  GVL_CAM.Control[nAxis].MotionFunction       := ADR(GVL_CAM.MotionFunction);
  GVL_CAM.Control[nAxis].MotionFunctionPoint  := ADR(GVL_CAM.MotionFunctionPoint);
END_FOR
//-----------------------------------------------------------------------------------------------------------------
// assign dataflow/
//-----------------------------------------------------------------------------------------------------------------
//-----------------------------------------------------------------------------------------------------------------
// /INIT
//-----------------------------------------------------------------------------------------------------------------
CASE eInit
OF
  E_PROGRESS.PROGRESS_INVALID:
    FOR nAxis := 1 TO PLC_CONSTANT.MAX_AXIS
    DO
      GVL_MSG_AXIS.MessageLevelAxisCam[nAxis] := E_MessageType.eMessageVerbose;//GVL_MSG.MessageLevel;
    END_FOR
    nAxisInit                                 := 1;
    eInit                                     := E_PROGRESS.PROGRESS_INIT;
  //-----------------------------------------------------------------------------
  //-----------------------------------------------------------------------------
  E_PROGRESS.PROGRESS_INIT:
    stMsg.eType                               := E_MessageType.eMessageInfo;
    stMsg.eDevice                             := e_Device.Device_Main;
    stMsg.eSubdevice                          := e_SubDevice.MainInit;
    stMsg.iErrorNumber                        := MAX_AXIS;
    stMsg.sText                               := concat('CAM.eInit: ', TO_STRING(eInit));
    f_MessageSet(stMsg);

    eInit                                     := E_PROGRESS.PROGRESS_BUSY;
  //-----------------------------------------------------------------------------
  //-----------------------------------------------------------------------------
  E_PROGRESS.PROGRESS_BUSY:
    eInit                                     := E_PROGRESS.PROGRESS_PREPARE;
  //-----------------------------------------------------------------------------
  //-----------------------------------------------------------------------------
  E_PROGRESS.PROGRESS_PREPARE:
    stMsg.eType                               := E_MessageType.eMessageVerbose;
    stMsg.eDevice                             := e_Device.Camming;
    stMsg.eSubdevice                          := e_SubDevice.CamStartUp;
    stMsg.iErrorNumber                        := nAxisInit;
    stMsg.sText                               := concat('AxisInit: ', TO_STRING(nAxisInit));

    IF (GVL_MSG_AXIS.MessageLevelAxisCam[nAxisInit] = E_MessageType.eMessageVerbose)
    THEN
      f_MessageSet(stMsg);
    END_IF

    GVL_CAM.Ctrl[nAxisInit].eCmd              := E_AXIS_CTRL.AXIS_NULL;
    eInit                                     := E_PROGRESS.PROGRESS_STARTUP;


  E_PROGRESS.PROGRESS_STARTUP:
    GVL_CAM.Ctrl[nAxisInit].eCmd              := E_AXIS_CTRL.AXIS_INIT;

    IF (GVL_CAM.State[nAxisInit].eState = E_AXIS_STATE.AXIS_INIT + E_PROGRESS.PROGRESS_ERROR)
    THEN
      eInit                                   := E_PROGRESS.PROGRESS_ERROR;

      stMsg.eType                             := E_MessageType.eMessageError;
      stMsg.eDevice                           := e_Device.Camming;
      stMsg.eSubdevice                        := e_SubDevice.CamStartUp;
      stMsg.iErrorNumber                      := nAxisInit;

      stMsg.sText                             := concat('CAM.eInit ERROR at Index: ', TO_STRING(nAxisInit));
      f_MessageSet(stMsg);

    ELSIF (GVL_CAM.State[nAxisInit].eState = E_AXIS_STATE.AXIS_INIT + E_PROGRESS.PROGRESS_DONE)
    THEN
      eInit                                   := E_PROGRESS.PROGRESS_CHECK;
    END_IF


  E_PROGRESS.PROGRESS_CHECK:
    IF (nAxisInit > PLC_CONSTANT.MAX_AXIS-1)
    THEN
      eInit                                   := E_PROGRESS.PROGRESS_DONE;

      stMsg.eType                             := E_MessageType.eMessageInfo;
      stMsg.eDevice                           := e_Device.Device_Cam;
      stMsg.eSubdevice                        := e_SubDevice.CamStartUp;
      stMsg.iErrorNumber                      := MAX_AXIS;

      stMsg.sText                             := concat('CAM.eInit: ', TO_STRING(eInit));
      f_MessageSet(stMsg);

      FOR nAxis := 1 TO PLC_CONSTANT.MAX_AXIS
      DO
        GVL_MSG_AXIS.MessageLevelAxisCam[nAxis]  := GVL_MSG_AXIS.MessageLevel;
      END_FOR
    ELSE
      nAxisInit                               := nAxisInit + 1;
      eInit                                   := E_PROGRESS.PROGRESS_PREPARE;
    END_IF
END_CASE
//-----------------------------------------------------------------------------------------------------------------
// INIT
//-----------------------------------------------------------------------------------------------------------------
//-----------------------------------------------------------------------------------------------------------------
// /cyclic
//-----------------------------------------------------------------------------------------------------------------
IF (eInit <> E_PROGRESS.PROGRESS_ERROR)
THEN
  FOR nAxis := 1 TO PLC_CONSTANT.MAX_AXIS
  DO
      GVL_CAM.Control[nAxis].Cycle();
  END_FOR
END_IF
//-----------------------------------------------------------------------------------------------------------------
// cyclic/
//-----------------------------------------------------------------------------------------------------------------

END_PROGRAM

// ---- PLC_MOTION/NCI/class/FB_NciChannelCtrl.TcPOU
(*
-------------------------------------------------------------------------------
	NCI Channel Control

  2020/05/20  HAUD  0.1     kinematic and NCI separation
  2022/10/22  HAUD  0.2     PLC_OPEN_DRIVE adaption
  2023/12/29  HAUD  0.3     PLC_STATE_DRIVE adaption
-------------------------------------------------------------------------------
*)

// This SOFTWARE is provided as an Exemple by THE PROVIDER "as is" and "with all faults." THE PROVIDER makes no 
// representations or warranties of any kind concerning the safety, suitability, lack of viruses, inaccuracies, 
// typographical errors, or other harmful components of this SOFTWARE. There are inherent dangers in the use of 
// any software, and you are solely responsible for determining whether this SOFTWARE is compatible with your 
// equipment and other software installed on your equipment. You are also solely responsible for the protection 
// of your equipment and backup of your data, and THE PROVIDER will not be liable for any damages you may suffer 
// in connection with using, modifying, or distributing this SOFTWARE.

FUNCTION_BLOCK FB_NciChannelCtrl EXTENDS FB_NciChannel IMPLEMENTS I_Nci_Ctrl
VAR
  _stChannelRef         : ST_NciChannel_Ref;
  _nChnId               : UINT;

  _eCtrl,
  _eCtrlOld             : E_NCI_CTRL;

  _eState               : E_NCI_STATE;

  _eInit,
  _eResult,
  _eResultOld           : E_PROGRESS;

  // control and state struct from outside world
  _Ctrl                 : POINTER TO ST_NCI_CTRL;
  _State                : POINTER TO ST_NCI_STATE;

  // M function to fetch for scope/debugging
  _MFuncScope           : POINTER TO ST_NCI_M_FUNC;

  _fPathVelo            : LREAL;
  _nBlockNo             : UDINT;
  _sProgLine            : STRING(100); 
  _nMFunc               : INT;
  _nStateItp            : UINT;
END_VAR

METHOD Check : BOOL
VAR_INST
 
END_VAR

IF NOT SUPER^.Check() THEN RETURN; END_IF

IF NOT (_Ctrl <> 0)
THEN
  _eCheck                     := E_CHECK_STATE.NCI_CTRL_POINTER_INVALID;
  RETURN;
END_IF

IF NOT (_State <> 0)
THEN
  _eCheck                     := E_CHECK_STATE.NCI_STATE_POINTER_INVALID;
  RETURN;
END_IF

IF NOT (_MFuncScope <> 0)
THEN
  _eCheck                     := E_CHECK_STATE.NCI_M_FUNC_POINTER_INVALID;
  RETURN;
END_IF

_eCheck                       := E_CHECK_STATE.CHECK_DONE;
Check                         := TRUE;
END_METHOD

PROPERTY ChnCtrl : pointer to ST_NCI_CTRL
SET
_Ctrl := ChnCtrl;
END_SET
END_PROPERTY

PROPERTY ChnId : udint
GET
ChnId := _NciChannelRef^.NcToPlc.ChnId;
END_GET
END_PROPERTY

PROPERTY ChnState : pointer to ST_NCI_STATE
SET
_State := ChnState;
END_SET
END_PROPERTY

//
//  Cmd
//    - gets state for ctrl
//    - prepare your commands here
//    - init what you have to here
//
//-------------------------------------------------------------------------------------
METHOD PRIVATE Cmd  : E_NCI_STATE
VAR_INPUT
  eCmd      : E_NCI_CTRL;
END_VAR
VAR_INST
  _estate   : E_NCI_STATE;
  _stMsg    : ST_Message;
END_VAR

CASE eCmd
OF
  E_NCI_CTRL.INIT:
    // check axis configuration, clear group, reset Itp
    _eInit := _eResult      := Ctrl_Init(FALSE);
    _eState                 := E_NCI_STATE.INIT;
ELSE
  IF NOT (_eInit = E_PROGRESS.PROGRESS_DONE)
  THEN
    _eResult                := E_PROGRESS.PROGRESS_ERROR;
  
    _stMsg.eType            := E_MessageType.eMessageError;
    _stMsg.eDevice          := E_Device.NciChannelCtrl + (ChnId);
    _stMsg.eSubdevice       := e_Subdevice.NciControl;
    _stMsg.iErrorNumber     := 1;
  
    _stMsg.sText          := 'eInit:';
    _stMsg.sText          := concat(_stMsg.sText, TO_STRING(_eInit));
    _stMsg.sText          := concat(_stMsg.sText, ': ');
    _stMsg.sText          := concat(_stMsg.sText, TO_STRING(_eResult));

    f_MessageSet(_stMsg);

  ELSE
    CASE eCmd
    OF
      E_NCI_CTRL.IDLE:
        _eResult                := Ctrl_Idle(FALSE);
        _eState                 := E_NCI_STATE.IDLE;
    
      E_NCI_CTRL.FEED_TABLE:
        // nothing implemented yet
        _eResult                := E_PROGRESS.PROGRESS_NOT_EXIST;
        _eState                 := E_NCI_STATE.FEED_TABLE;
    
      E_NCI_CTRL.RESET:
        _eResult                := Ctrl_Reset(FALSE);
        _eState                 := E_NCI_STATE.RESET;
    
      E_NCI_CTRL.LOAD_PROG:
        _eResult                := Ctrl_LoadProg(FALSE);
        _eState                 := E_NCI_STATE.LOAD_PROG;
    
      E_NCI_CTRL.BUILD_GROUP:
        _eResult                := Ctrl_BuildGroup(FALSE);
        _eState                 := E_NCI_STATE.BUILD_GROUP;
    
      E_NCI_CTRL.CLEAR_GROUP:
        _eResult                := Ctrl_ClearGroup(FALSE);
        _eState                 := E_NCI_STATE.CLEAR_GROUP;
    
      E_NCI_CTRL.START:
        _eResult                := Ctrl_Start(FALSE);
        _eState                 := E_NCI_STATE.START;
    
      E_NCI_CTRL.STOP:
        _eResult                := Ctrl_Stop(FALSE);
        _eState                 := E_NCI_STATE.STOP;
    
      E_NCI_CTRL.STO_STOP:
        _eResult                := Ctrl_Stop_STO(FALSE);
        _eState                 := E_NCI_STATE.STO_STOP;
    
      E_NCI_CTRL.RESTART_STEP_ON:
        _eResult                := Ctrl_Restart(FALSE);
        _eState                 := E_NCI_STATE.RESTART_STEP_ON;
    
      E_NCI_CTRL.M_FUNC_QUIT:
        _eResult                := Ctrl_ConfirmHsk(FALSE);
        _eState                 := E_NCI_STATE.M_FUNC_QUIT;
    
      E_NCI_CTRL.READ_R_PARA:
        _eResult                := Ctrl_R_Parameter_Rd(FALSE);
        _eState                 := E_NCI_STATE.READ_R_PARA;
    
      E_NCI_CTRL.WRITE_R_PARA:
        _eResult                := Ctrl_R_Parameter_Wrt(FALSE);
        _eState                 := E_NCI_STATE.WRITE_R_PARA;
    ELSE
      _eState                 := E_NCI_STATE.NULL;
  
      IF (eCmd = E_NCI_CTRL.NULL)
      THEN
        _eResult              := E_PROGRESS.PROGRESS_DONE;
      ELSE
        _eResult              := E_PROGRESS.PROGRESS_INVALID;
  
        _stMsg.eType          := E_MessageType.eMessageError;
        _stMsg.eDevice        := E_Device.NciChannelCtrl + (ChnId);
        _stMsg.eSubdevice     := e_Subdevice.NciControl;
        _stMsg.iErrorNumber   := 0;
  
        _stMsg.sText          := 'E_NCI_CTRL.';
        _stMsg.sText          := concat(_stMsg.sText, TO_STRING(eCmd));
        _stMsg.sText          := concat(_stMsg.sText, ': ');
        _stMsg.sText          := concat(_stMsg.sText, TO_STRING(_eResult));
  
        f_MessageSet(_stMsg);
      END_IF
    END_CASE
  END_IF
END_CASE


Cmd                         := _eState;
END_METHOD

METHOD PRIVATE Ctrl_BuildGroup : E_PROGRESS
VAR_INPUT
  Execute           : BOOL;
END_VAR
VAR_INST
  _eJobResult,
  _eState           : E_PROGRESS;
END_VAR
IF NOT Check() THEN Ctrl_BuildGroup := E_PROGRESS.PROGRESS_ERROR; RETURN; END_IF
IF NOT Execute THEN _eState := E_PROGRESS.PROGRESS_INIT; END_IF

CASE _eState
OF
  E_PROGRESS.PROGRESS_INIT:
    IF Execute 
    THEN
      _eJobResult                   := BuilDGroup(FALSE);
      _eState                       := E_PROGRESS.PROGRESS_BUSY;
    END_IF
END_CASE
CASE _eState
OF
  E_PROGRESS.PROGRESS_BUSY:
    _eJobResult                     := BuilDGroup(TRUE);

    IF (_eJobResult = E_PROGRESS.PROGRESS_ERROR)
    THEN
      BuilDGroup(FALSE);
      _eState                       := E_PROGRESS.PROGRESS_ERROR;

    ELSIF (_eJobResult = E_PROGRESS.PROGRESS_DONE)
    THEN
      BuilDGroup(FALSE);
      _eState                       := E_PROGRESS.PROGRESS_STARTUP;
    END_IF
END_CASE
CASE _eState
OF
  E_PROGRESS.PROGRESS_STARTUP:
    _eState                         := E_PROGRESS.PROGRESS_PREPARE;
END_CASE
CASE _eState
OF
  E_PROGRESS.PROGRESS_PREPARE:
    _eState                         := E_PROGRESS.PROGRESS_CHECK;
END_CASE
CASE _eState
OF
  E_PROGRESS.PROGRESS_CHECK:
    _eState                         := E_PROGRESS.PROGRESS_OCCUPIED;
END_CASE
CASE _eState
OF
  E_PROGRESS.PROGRESS_OCCUPIED:
    _eState                         := E_PROGRESS.PROGRESS_WORKING;
END_CASE
CASE _eState
OF
  E_PROGRESS.PROGRESS_WORKING:
    _eState                         := E_PROGRESS.PROGRESS_DONE;
END_CASE

Ctrl_BuildGroup                      := _eState;
END_METHOD

METHOD PRIVATE Ctrl_ClearGroup : E_PROGRESS
VAR_INPUT
  Execute           : BOOL;
END_VAR
VAR_INST
  _eJobResult,
  _eState           : E_PROGRESS;
END_VAR
IF NOT Check() THEN Ctrl_ClearGroup := E_PROGRESS.PROGRESS_ERROR; RETURN; END_IF
IF NOT Execute THEN _eState := E_PROGRESS.PROGRESS_INIT; END_IF

CASE _eState
OF
  E_PROGRESS.PROGRESS_INIT:
    IF Execute 
    THEN
      _eJobResult                           := ClearGroup(FALSE);
      _eState                               := E_PROGRESS.PROGRESS_BUSY;
    END_IF

  E_PROGRESS.PROGRESS_BUSY:
    _eJobResult                             := ClearGroup(TRUE);
    IF (_eJobResult = E_PROGRESS.PROGRESS_ERROR)
    THEN
      ClearGroup(FALSE);
      _eState                               := E_PROGRESS.PROGRESS_ERROR;

    ELSIF (_eJobResult = E_PROGRESS.PROGRESS_DONE)
    THEN
      ClearGroup(FALSE);
      _eJobResult                           := ItpReset(FALSE);
      _eState                               := E_PROGRESS.PROGRESS_STARTUP;
    END_IF

  E_PROGRESS.PROGRESS_STARTUP:
    _eJobResult                             := ItpReset(TRUE);
    IF (_eJobResult = E_PROGRESS.PROGRESS_ERROR)
    THEN
      ItpReset(FALSE);
      _eState                               := E_PROGRESS.PROGRESS_ERROR;

    ELSIF (_eJobResult = E_PROGRESS.PROGRESS_DONE)
    THEN
      ItpReset(FALSE);
      _eState                               := E_PROGRESS.PROGRESS_PREPARE;
    END_IF

  E_PROGRESS.PROGRESS_PREPARE:
    IF (_NciChannelRef^.NcToPlc.HskMFuncReq = 0)
    THEN
      _eState                               := E_PROGRESS.PROGRESS_DONE;
    ELSE
      _NciChannelRef^.PlcToNc.MFuncGranted  := 0;
      _eState                               := E_PROGRESS.PROGRESS_CHECK;
    END_IF

  E_PROGRESS.PROGRESS_CHECK:
      _NciChannelRef^.PlcToNc.MFuncGranted  := 1;
      _eState                               := E_PROGRESS.PROGRESS_PREPARE;

  E_PROGRESS.PROGRESS_DONE:
    _NciChannelRef^.PlcToNc.MFuncGranted    := 0;
END_CASE


Ctrl_ClearGroup                             := _eState;
END_METHOD

METHOD PRIVATE Ctrl_ConfirmHsk : E_PROGRESS
VAR_INPUT
  Execute           : BOOL;
END_VAR
VAR_INST
  _eJobResult,
  _eState           : E_PROGRESS;
END_VAR
IF NOT Check() THEN Ctrl_ConfirmHsk := E_PROGRESS.PROGRESS_ERROR; RETURN; END_IF
IF NOT Execute THEN _eState := E_PROGRESS.PROGRESS_INIT; END_IF

CASE _eState
OF
  E_PROGRESS.PROGRESS_INIT:
    IF Execute 
    THEN
      _eJobResult                         := ConfirmHSK(FALSE);
      _eState                             := E_PROGRESS.PROGRESS_BUSY;
    END_IF
END_CASE
CASE _eState
OF

  E_PROGRESS.PROGRESS_BUSY:
    _eJobResult                           := ConfirmHSK(TRUE);

    IF (_eJobResult = E_PROGRESS.PROGRESS_ERROR)
    THEN
      ConfirmHSK(FALSE);
      _eState                             := E_PROGRESS.PROGRESS_ERROR;

    ELSIF (_eJobResult = E_PROGRESS.PROGRESS_DONE)
    THEN
      ConfirmHSK(FALSE);
      _eState                             := E_PROGRESS.PROGRESS_PREPARE;
    END_IF
END_CASE
CASE _eState
OF
  E_PROGRESS.PROGRESS_PREPARE:
    _eState                               := E_PROGRESS.PROGRESS_DONE;
    // update connected struct data
    _MFuncScope^.FastMFuncMask            := _NciChannelRef^.NcToPlc.FastMFuncMask;
    _MFuncScope^.HskMFuncNo               := _NciChannelRef^.NcToPlc.HskMFuncNo;
    _MFuncScope^.HskMFuncReq              := _NciChannelRef^.NcToPlc.HskMFuncReq;
    _MFuncScope^.HFuncValue               := _NciChannelRef^.NcToPlc.HFuncValue;
    _MFuncScope^.MFuncGranted             := _NciChannelRef^.PlcToNc.MFuncGranted;
END_CASE

Ctrl_ConfirmHsk                            := _eState;
END_METHOD

METHOD PRIVATE Ctrl_Idle : E_PROGRESS
VAR_INPUT
  Execute           : BOOL;
END_VAR
VAR_INST
  _eJobResult,
  _eState           : E_PROGRESS;

  _nErr             : DWORD;
  _NciAxisIds       : ARRAY[1..8] OF DWORD;

  _stMsg            : ST_Message;
END_VAR
IF NOT Check() THEN Ctrl_Idle := E_PROGRESS.PROGRESS_ERROR; RETURN; END_IF
IF NOT Execute THEN _eState := E_PROGRESS.PROGRESS_INIT; END_IF

CASE _eState
OF
  E_PROGRESS.PROGRESS_INIT:
    IF Execute 
    THEN
      _eJobResult                         := ItpReset(FALSE);
      _eState                             := E_PROGRESS.PROGRESS_BUSY;
    END_IF
END_CASE
CASE _eState
OF
  E_PROGRESS.PROGRESS_BUSY:
    IF (_NciChannelRef^.NcToPlc.ItpState <> Tc2_NCI.NCI_INTERPRETER_IDLE)
    THEN
      _eState                             := E_PROGRESS.PROGRESS_STARTUP;
    ELSE
      IF (_NciChannelRef^.PlcToNc.ChnAxesOvr > 0) AND NOT
         (_NciChannelRef^.NcToPlc.ChnState.8)
      THEN
        _eState                           := E_PROGRESS.PROGRESS_PREPARE;
      END_IF
    END_IF
END_CASE
CASE _eState
OF
  E_PROGRESS.PROGRESS_STARTUP:
    _eJobResult                           := ItpReset(TRUE);
    IF (_eJobResult = E_PROGRESS.PROGRESS_ERROR)
    THEN
      ItpReset(FALSE);
      _eState                             := E_PROGRESS.PROGRESS_ERROR;

    ELSIF (_eJobResult = E_PROGRESS.PROGRESS_DONE)
    THEN
      ItpReset(FALSE);
      _eState                             := E_PROGRESS.PROGRESS_PREPARE;
    END_IF

  E_PROGRESS.PROGRESS_PREPARE:
    _NciChannelRef^.PlcToNc.MFuncGranted  := 0;
    _eState                               := E_PROGRESS.PROGRESS_CHECK;

END_CASE
CASE _eState
OF
  E_PROGRESS.PROGRESS_CHECK:
    _nErr                                 := ItpGetGroupAxisIds(_NciAxisIds, _NciChannelRef^.NcToPlc);

    IF (_NciChannelRef^.NcToPlc.HskMFuncReq = 0)
    THEN
      IF (_nErr <> 0)
      THEN
        _eState                           := E_PROGRESS.PROGRESS_ERROR;
        _stMsg.eType                      := E_MessageType.eMessageError;
        _stMsg.eDevice                    := ChannelDevice;
        _stMsg.eSubdevice                 := e_Subdevice.NciIdle;
        _stMsg.iErrorNumber               := _nErr;
        _stMsg.sText                      := concat('ItpGetGroupAxisIds Error: ', TO_STRING(_nErr));

        f_MessageSet(_stMsg);
      ELSE
        _eState                           := E_PROGRESS.PROGRESS_DONE;
      END_IF
    ELSE
      _eState                             := E_PROGRESS.PROGRESS_STARTUP;
    END_IF
END_CASE

Ctrl_Idle                                := _eState;
END_METHOD

METHOD Ctrl_Init : E_PROGRESS
VAR_INPUT
  Execute           : BOOL;
END_VAR
VAR_INST
  _eJobResult,
  _eState           : E_PROGRESS;
  _rValue           : LREAL;
  _udiErr           : UDINT;

  _nErr             : DWORD;
  _NciAxisIds       : ARRAY[1..8] OF DWORD;

  _stMsg            : ST_Message;
END_VAR
IF NOT Check() THEN _eState := E_PROGRESS.PROGRESS_ERROR; END_IF
IF NOT Execute THEN _eState := E_PROGRESS.PROGRESS_INIT; END_IF

CASE _eState
OF
  E_PROGRESS.PROGRESS_INIT:
    IF Execute 
    THEN
      memset(ADR(_stMsg),0,SIZEOF(_stMsg));
      _udiErr                       := 0;
      _rValue                       := 0;
      _eState                       := E_PROGRESS.PROGRESS_BUSY;
    END_IF
END_CASE
CASE _eState
OF
  E_PROGRESS.PROGRESS_BUSY:
    IF NOT (_stCfgAxes^.nXAxisId > 0) OR
       NOT (_stCfgAxes^.nYAxisId > 0) OR
       NOT (_stCfgAxes^.nZAxisId > 0)
    THEN
      _eState                       := E_PROGRESS.PROGRESS_OCCUPIED;

      _stMsg.eType                  := E_MessageType.eMessageWarning;
      _stMsg.eDevice                := ChannelDevice;
      _stMsg.eSubdevice             := e_Subdevice.NciStartUp;
      _stMsg.iErrorNumber           := _eState;
      _stMsg.sText                  := concat('Init NCI channel AxisConfig: ', TO_STRING(_eState));

      f_MessageSet(_stMsg);
    ELSE
      _eJobResult                   := ItpReset(FALSE);
      _eState                       := E_PROGRESS.PROGRESS_STARTUP;
    END_IF
END_CASE
CASE _eState
OF
  E_PROGRESS.PROGRESS_STARTUP:
    _eJobResult                     := ItpReset(TRUE);
    IF (_eJobResult = E_PROGRESS.PROGRESS_ERROR)
    THEN
      _eState                       := E_PROGRESS.PROGRESS_ERROR;
    ELSIF (_eJobResult = E_PROGRESS.PROGRESS_DONE)
    THEN
      _eJobResult                   := ItpReset  (FALSE);
      _eJobResult                   := ClearGroup(FALSE);
      _eState                       := E_PROGRESS.PROGRESS_PREPARE;
    END_IF
END_CASE
CASE _eState
OF
  E_PROGRESS.PROGRESS_PREPARE:
    _eJobResult                     := ClearGroup(TRUE);
    IF (_eJobResult = E_PROGRESS.PROGRESS_ERROR)
    THEN
      _eState                       := E_PROGRESS.PROGRESS_ERROR;
    ELSIF (_eJobResult = E_PROGRESS.PROGRESS_DONE)
    THEN
      _eJobResult                   := ClearGroup(FALSE);
      _eState                       := E_PROGRESS.PROGRESS_CHECK;
    END_IF

END_CASE
CASE _eState
OF
  E_PROGRESS.PROGRESS_CHECK:
    _eState                         := E_PROGRESS.PROGRESS_WORKING;
END_CASE
CASE _eState
OF
  E_PROGRESS.PROGRESS_OCCUPIED:
    IF (_stCfgAxes^.nXAxisId > 0) AND
       (_stCfgAxes^.nYAxisId > 0) AND
       (_stCfgAxes^.nZAxisId > 0)
    THEN
      _eState                       := E_PROGRESS.PROGRESS_STARTUP;

      _stMsg.eType                  := E_MessageType.eMessageInfo;
      _stMsg.eDevice                := ChannelDevice;
      _stMsg.eSubdevice             := e_Subdevice.NciStartUp;
      _stMsg.iErrorNumber           := _eState;
      _stMsg.sText                  := concat('Init NCI channel AxisConfig: ', TO_STRING(_eState));

      IF (_MessageLevel < E_MessageType.eMessageError)
      THEN
        f_MessageSet(_stMsg);
      END_IF
    END_IF
END_CASE
CASE _eState
OF
  E_PROGRESS.PROGRESS_WORKING:
    _eState                         := E_PROGRESS.PROGRESS_DONE;
END_CASE

Ctrl_Init                           := _eState;
END_METHOD

METHOD PRIVATE Ctrl_LoadProg : E_PROGRESS
VAR_INPUT
  Execute           : BOOL;
END_VAR
VAR_INST
  _eJobResult,
  _eState           : E_PROGRESS;
END_VAR
IF NOT Check() THEN Ctrl_LoadProg := E_PROGRESS.PROGRESS_ERROR; RETURN; END_IF
IF NOT Execute THEN _eState := E_PROGRESS.PROGRESS_INIT; END_IF

CASE _eState
OF
  E_PROGRESS.PROGRESS_INIT:
    IF Execute 
    THEN
      _eJobResult                         := LoadProg(FALSE);
      _eState                             := E_PROGRESS.PROGRESS_BUSY;
    END_IF

  E_PROGRESS.PROGRESS_BUSY:
    _NciChannelRef^.PlcToNc.MFuncGranted  := 0;
    _eJobResult                           := LoadProg(TRUE);

    IF (_eJobResult = E_PROGRESS.PROGRESS_ERROR)
    THEN
      LoadProg(FALSE);
      _eState                             := E_PROGRESS.PROGRESS_ERROR;

    ELSIF (_eJobResult = E_PROGRESS.PROGRESS_DONE)
    THEN
      LoadProg(FALSE);
      _eState                             := E_PROGRESS.PROGRESS_DONE;
    END_IF
END_CASE

Ctrl_LoadProg                      := _eState;
END_METHOD

METHOD PRIVATE Ctrl_R_Parameter_Rd : E_PROGRESS
VAR_INPUT
  Execute           : BOOL;
END_VAR
VAR_INST
  _eJobResult,
  _eState           : E_PROGRESS;
END_VAR
IF NOT Check() THEN Ctrl_R_Parameter_Rd := E_PROGRESS.PROGRESS_ERROR; RETURN; END_IF
IF NOT Execute THEN _eState := E_PROGRESS.PROGRESS_INIT; END_IF

CASE _eState
OF
  E_PROGRESS.PROGRESS_INIT:
    IF Execute 
    THEN
      _eJobResult                         := ReadRParams(FALSE);
      _eState                             := E_PROGRESS.PROGRESS_BUSY;
    END_IF

  E_PROGRESS.PROGRESS_BUSY:
    _NciChannelRef^.PlcToNc.MFuncGranted  := 0;
    _eJobResult                           := ReadRParams(TRUE);

    IF (_eJobResult = E_PROGRESS.PROGRESS_ERROR)
    THEN
      ReadRParams(FALSE);
      _eState                             := E_PROGRESS.PROGRESS_ERROR;

    ELSIF (_eJobResult = E_PROGRESS.PROGRESS_DONE)
    THEN
      ReadRParams(FALSE);
      _eState                             := E_PROGRESS.PROGRESS_STARTUP;
    END_IF
END_CASE
CASE _eState
OF
  E_PROGRESS.PROGRESS_STARTUP:
    _NciChannelRef^.PlcToNc.MFuncGranted  := 1;
    _eState                               := E_PROGRESS.PROGRESS_PREPARE;

  E_PROGRESS.PROGRESS_PREPARE:
    _NciChannelRef^.PlcToNc.MFuncGranted  := 0;
    _eState                               := E_PROGRESS.PROGRESS_DONE;
END_CASE

Ctrl_R_Parameter_Rd                       := _eState;
END_METHOD

METHOD PRIVATE Ctrl_R_Parameter_Wrt : E_PROGRESS
VAR_INPUT
  Execute           : BOOL;
END_VAR
VAR_INST
  _eJobResult,
  _eState           : E_PROGRESS;
END_VAR
IF NOT Check() THEN Ctrl_R_Parameter_Wrt := E_PROGRESS.PROGRESS_ERROR; RETURN; END_IF
IF NOT Execute THEN _eState := E_PROGRESS.PROGRESS_INIT; END_IF

CASE _eState
OF
  E_PROGRESS.PROGRESS_INIT:
    IF Execute 
    THEN
      _eJobResult                         := WriteRParams(FALSE);
      _eState                             := E_PROGRESS.PROGRESS_BUSY;
    END_IF

  E_PROGRESS.PROGRESS_BUSY:
    _NciChannelRef^.PlcToNc.MFuncGranted  := 0;
    _eJobResult                           := WriteRParams(TRUE);

    IF (_eJobResult = E_PROGRESS.PROGRESS_ERROR)
    THEN
      WriteRParams(FALSE);
      _eState                             := E_PROGRESS.PROGRESS_ERROR;

    ELSIF (_eJobResult = E_PROGRESS.PROGRESS_DONE)
    THEN
      WriteRParams(FALSE);
      _eState                             := E_PROGRESS.PROGRESS_STARTUP;
    END_IF
END_CASE
CASE _eState
OF
  E_PROGRESS.PROGRESS_STARTUP:
    _NciChannelRef^.PlcToNc.MFuncGranted  := 1;
    _eState                               := E_PROGRESS.PROGRESS_PREPARE;

  E_PROGRESS.PROGRESS_PREPARE:
    _NciChannelRef^.PlcToNc.MFuncGranted  := 0;
    _eState                               := E_PROGRESS.PROGRESS_DONE;
END_CASE

Ctrl_R_Parameter_Wrt                      := _eState;
END_METHOD

METHOD PRIVATE Ctrl_Reset : E_PROGRESS
VAR_INPUT
  Execute           : BOOL;
END_VAR
VAR_INST
  _eJobResult,
  _eState           : E_PROGRESS;
END_VAR
IF NOT Check() THEN Ctrl_Reset := E_PROGRESS.PROGRESS_ERROR; RETURN; END_IF
IF NOT Execute THEN _eState := E_PROGRESS.PROGRESS_INIT; END_IF

CASE _eState
OF
  E_PROGRESS.PROGRESS_INIT:
    IF Execute 
    THEN
      _eJobResult                         := ItpReset(FALSE);
      _eState                             := E_PROGRESS.PROGRESS_BUSY;
    END_IF
END_CASE
CASE _eState
OF
  E_PROGRESS.PROGRESS_BUSY:
    _NciChannelRef^.PlcToNc.MFuncGranted  := 0;
    _eJobResult                           := ItpReset(TRUE);

    IF (_eJobResult = E_PROGRESS.PROGRESS_ERROR)
    THEN
      ItpReset(FALSE);
      _eState                             := E_PROGRESS.PROGRESS_ERROR;

    ELSIF (_eJobResult = E_PROGRESS.PROGRESS_DONE)
    THEN
      ItpReset(FALSE);
      _eState                             := E_PROGRESS.PROGRESS_STARTUP;
    END_IF

  E_PROGRESS.PROGRESS_STARTUP:
    _NciChannelRef^.PlcToNc.MFuncGranted  := 1;
    _eState                               := E_PROGRESS.PROGRESS_PREPARE;

  E_PROGRESS.PROGRESS_PREPARE:
    _NciChannelRef^.PlcToNc.MFuncGranted  := 0;
    _eState                               := E_PROGRESS.PROGRESS_CHECK;

END_CASE
CASE _eState
OF
  E_PROGRESS.PROGRESS_CHECK:
    IF (_NciChannelRef^.NcToPlc.HskMFuncReq = 0)
    THEN
      _eState                             := E_PROGRESS.PROGRESS_DONE;
    ELSE
      _eState                             := E_PROGRESS.PROGRESS_STARTUP;
    END_IF
END_CASE

Ctrl_Reset                                := _eState;
END_METHOD

METHOD PRIVATE Ctrl_Restart : E_PROGRESS
VAR_INPUT
  Execute           : BOOL;
END_VAR
VAR_INST
  _eJobResult,
  _eState           : E_PROGRESS;
END_VAR
IF NOT Check() THEN Ctrl_Restart := E_PROGRESS.PROGRESS_ERROR; RETURN; END_IF
IF NOT Execute THEN _eState := E_PROGRESS.PROGRESS_INIT; END_IF

CASE _eState
OF
  E_PROGRESS.PROGRESS_INIT:
    IF Execute 
    THEN
      _eJobResult                         := StepOnAfterEStop(FALSE);
      _eState                             := E_PROGRESS.PROGRESS_BUSY;
    END_IF
END_CASE
CASE _eState
OF
  E_PROGRESS.PROGRESS_BUSY:
    _NciChannelRef^.PlcToNc.MFuncGranted  := 0;
    _eJobResult                           := StepOnAfterEStop(TRUE);

    IF (_eJobResult = E_PROGRESS.PROGRESS_ERROR)
    THEN
      StepOnAfterEStop(FALSE);
      _eState                             := E_PROGRESS.PROGRESS_ERROR;

    ELSIF (_eJobResult = E_PROGRESS.PROGRESS_DONE)
    THEN
      StepOnAfterEStop(FALSE);
      _eState                             := E_PROGRESS.PROGRESS_DONE;
    END_IF
END_CASE


Ctrl_Restart                              := _eState;
END_METHOD

METHOD PRIVATE Ctrl_Start : E_PROGRESS
VAR_INPUT
  Execute           : BOOL;
END_VAR
VAR_INST
  _eJobResult,
  _eState           : E_PROGRESS;
END_VAR
IF NOT Check() THEN Ctrl_Start := E_PROGRESS.PROGRESS_ERROR; RETURN; END_IF
IF NOT Execute THEN _eState := E_PROGRESS.PROGRESS_INIT; END_IF

CASE _eState
OF
  E_PROGRESS.PROGRESS_INIT:
    IF Execute 
    THEN
      _eJobResult                         := StartStop(FALSE, TRUE, FALSE);
      _eState                             := E_PROGRESS.PROGRESS_BUSY;
    END_IF
END_CASE
CASE _eState
OF
  E_PROGRESS.PROGRESS_BUSY:
    _NciChannelRef^.PlcToNc.MFuncGranted  := 0;
    _eJobResult                           := StartStop(TRUE, TRUE, FALSE);

    IF (_eJobResult = E_PROGRESS.PROGRESS_ERROR)
    THEN
      StartStop(FALSE, TRUE, FALSE);
      _eState                             := E_PROGRESS.PROGRESS_ERROR;

    ELSIF (_eJobResult = E_PROGRESS.PROGRESS_DONE)
    THEN
      StartStop(FALSE, TRUE, FALSE);
      _eState                             := E_PROGRESS.PROGRESS_DONE;
    END_IF
END_CASE

Ctrl_Start                                := _eState;
END_METHOD

METHOD PRIVATE Ctrl_Stop : E_PROGRESS
VAR_INPUT
  Execute           : BOOL;
END_VAR
VAR_INST
  _eJobResult,
  _eState           : E_PROGRESS;
END_VAR
IF NOT Check() THEN Ctrl_Stop := E_PROGRESS.PROGRESS_ERROR; RETURN; END_IF
IF NOT Execute THEN _eState := E_PROGRESS.PROGRESS_INIT; END_IF

CASE _eState
OF
  E_PROGRESS.PROGRESS_INIT:
    IF Execute 
    THEN
      _eJobResult                         := StartStop(FALSE, FALSE, TRUE);
      _eState                             := E_PROGRESS.PROGRESS_BUSY;
    END_IF
END_CASE
CASE _eState
OF
  E_PROGRESS.PROGRESS_BUSY:
    _NciChannelRef^.PlcToNc.MFuncGranted  := 0;
    _eJobResult                           := StartStop(TRUE, FALSE, TRUE);

    IF (_eJobResult = E_PROGRESS.PROGRESS_ERROR)
    THEN
      StartStop(FALSE, FALSE, TRUE);
      _eState                             := E_PROGRESS.PROGRESS_ERROR;

    ELSIF (_eJobResult = E_PROGRESS.PROGRESS_DONE)
    THEN
      StartStop(FALSE, FALSE, TRUE);
      _eState                             := E_PROGRESS.PROGRESS_DONE;
    END_IF
END_CASE

Ctrl_Stop                                := _eState;
END_METHOD

METHOD PRIVATE Ctrl_Stop_STO : E_PROGRESS
VAR_INPUT
  Execute           : BOOL;
END_VAR
VAR_INST
  _eJobResult,
  _eState           : E_PROGRESS;
END_VAR
IF NOT Check() THEN Ctrl_Stop_STO := E_PROGRESS.PROGRESS_ERROR; RETURN; END_IF
IF NOT Execute THEN _eState := E_PROGRESS.PROGRESS_INIT; END_IF

CASE _eState
OF
  E_PROGRESS.PROGRESS_INIT:
    IF Execute 
    THEN
      _eJobResult                         := EStop(FALSE);
      _eState                             := E_PROGRESS.PROGRESS_BUSY;
    END_IF
END_CASE
CASE _eState
OF
  E_PROGRESS.PROGRESS_BUSY:
    _NciChannelRef^.PlcToNc.MFuncGranted  := 0;
    _eJobResult                           := EStop(TRUE);

    IF (_eJobResult = E_PROGRESS.PROGRESS_ERROR)
    THEN
      EStop(FALSE);
      _eState                             := E_PROGRESS.PROGRESS_ERROR;

    ELSIF (_eJobResult = E_PROGRESS.PROGRESS_DONE)
    THEN
      EStop(FALSE);
      _eState                             := E_PROGRESS.PROGRESS_DONE;
    END_IF
END_CASE

Ctrl_Stop_STO                                := _eState;
END_METHOD

METHOD Cycle  : e_progress
VAR_INST
  _eCycle     : E_PROGRESS;
END_VAR
//-----------------------------------------------------------------------------
//-----------------------------------------------------------------------------
// cyclic pointer to NCI wrapper
//-----------------------------------------------------------------------------
ChannelRef    := ADR(_stChannelRef);
//-----------------------------------------------------------------------------
//-----------------------------------------------------------------------------
IF NOT Check() THEN Cycle := _eCycle := _eResult := E_PROGRESS.PROGRESS_ERROR; RETURN; END_IF
//-----------------------------------------------------------------------------
//-----------------------------------------------------------------------------
ChannelDevice := e_Device.NciChannel + TO_UINT(ChnId);
//-----------------------------------------------------------------------------
//-----------------------------------------------------------------------------
// cyclic data for M func from NCI interface
//-----------------------------------------------------------------------------
_MFuncScope^.FastMFuncMask    := _NciChannelRef^.NcToPlc.FastMFuncMask;
_MFuncScope^.HskMFuncNo       := _NciChannelRef^.NcToPlc.HskMFuncNo;
_MFuncScope^.HskMFuncReq      := _NciChannelRef^.NcToPlc.HskMFuncReq;
_MFuncScope^.HFuncValue       := _NciChannelRef^.NcToPlc.HFuncValue;
_MFuncScope^.MFuncGranted     := _NciChannelRef^.PlcToNc.MFuncGranted;
//-----------------------------------------------------------------------------
//-----------------------------------------------------------------------------
// M-Func to catch
//-----------------------------------------------------------------------------
IF HSK 
THEN
  _nMFunc := MFunc;
END_IF
//-----------------------------------------------------------------------------
//-----------------------------------------------------------------------------
_eCtrl                         := _Ctrl^.eCmd;
//-----------------------------------------------------------------------------
//-----------------------------------------------------------------------------
// cmd change
//-----------------------------------------------------------------------------
IF (_eCtrl <> _eCtrlOld)
THEN
  LogControl();
  _eState                     := Cmd(_eCtrl);
  _eCtrlOld                   := _eCtrl;
END_IF
//-----------------------------------------------------------------------------
//-----------------------------------------------------------------------------
CASE _eResult
OF
  E_PROGRESS.PROGRESS_INVALID:
    _State^.eState            := TO_UINT(E_PROGRESS.PROGRESS_ERROR);

  E_PROGRESS.PROGRESS_ERROR:
    _State^.eState            := _eState + E_PROGRESS.PROGRESS_ERROR;
    Cycle         := _eCycle  := E_PROGRESS.PROGRESS_ERROR;

  E_PROGRESS.PROGRESS_DONE:
    _State^.eState            := _eState + E_PROGRESS.PROGRESS_DONE;

ELSE
    _State^.eState            := _eState + _eResult;
    Cycle         := _eCycle  := E_PROGRESS.PROGRESS_WORKING;
  CASE _eState
  OF
  E_NCI_STATE.INIT:
    _eResult      := _eInit   := Ctrl_Init(TRUE);

  E_NCI_STATE.IDLE:
    _eResult                  := Ctrl_Idle(TRUE);

  E_NCI_STATE.RESET:
    _eResult                  := Ctrl_Reset(TRUE);

  E_NCI_STATE.LOAD_PROG:
    _eResult                  := Ctrl_LoadProg(TRUE);

  E_NCI_STATE.BUILD_GROUP:
    _eResult                  := Ctrl_BuildGroup(TRUE);

  E_NCI_STATE.CLEAR_GROUP:
    _eResult                  := Ctrl_ClearGroup(TRUE);

  E_NCI_STATE.START:
    _eResult                  := Ctrl_Start(TRUE);

  E_NCI_STATE.STOP:
    _eResult                  := Ctrl_Stop(TRUE);

  E_NCI_STATE.STO_STOP:
    _eResult                  := Ctrl_Stop_STO(TRUE);

  E_NCI_STATE.RESTART_STEP_ON:
    _eResult                  := Ctrl_Restart(TRUE);

  E_NCI_STATE.M_FUNC_QUIT:
    _eResult                  := Ctrl_ConfirmHsk(TRUE);

  E_NCI_STATE.READ_R_PARA:
    _eResult                  := Ctrl_R_Parameter_Rd(TRUE);

  E_NCI_STATE.WRITE_R_PARA:
    _eResult                  := Ctrl_R_Parameter_Wrt(TRUE);
  END_CASE
END_CASE
//-----------------------------------------------------------------------------
//-----------------------------------------------------------------------------
//  OnChange of execution state result
//    - log result
//-----------------------------------------------------------------------------
IF (_eResult <> _eResultOld)
THEN
  LogResult();
  _eResultOld                 := _eResult;
END_IF
//-----------------------------------------------------------------------------
//-----------------------------------------------------------------------------
//  cyclic data from ChannelRef
//-----------------------------------------------------------------------------
_State^.rAxisOverride         := _NciChannelRef^.PlcToNc.ChnAxesOvr;
_State^.bMFuncReq             := TO_BOOL(_NciChannelRef^.NcToPlc.HskMFuncReq);
_State^.nMFunc                := _NciChannelRef^.NcToPlc.HskMFuncNo;
_State^.nItpState             := GetItpState();
//-----------------------------------------------------------------------------
//-----------------------------------------------------------------------------
END_METHOD

PROPERTY ItfChannel : I_NciChannel
GET
ItfChannel := SUPER^;
END_GET
END_PROPERTY

METHOD LogControl
VAR_INST
  _sResult,
  _sCtrl            : STRING(30);

  _stMsg            : ST_Message;
END_VAR
  _stMsg.eType               := E_MessageType.eMessageInfo;
  _stMsg.eDevice             := E_Device.NciChannelCtrl + TO_UINT(ChnId);
  _stMsg.eSubdevice          := e_Subdevice.NciControl;
  _stMsg.iErrorNumber        := 0;

  _sCtrl                     := concat('E_NCI_CTRL', '.');
  _sCtrl                     := concat(_sCtrl, TO_STRING(_eCtrl));

  _stMsg.sText               := concat('new command: ', _sCtrl);

  IF (_MessageLevel < E_MessageType.eMessageError)
  THEN
    f_MessageSet(_stMsg);
  ELSE
    IF (_stMsg.eType = E_MessageType.eMessageError)
    THEN
      f_MessageSet(_stMsg);
    END_IF
  END_IF
END_METHOD

METHOD PRIVATE LogResult
VAR_INST
  _sResult,
  _sCtrl            : STRING(30);

  _stMsg            : ST_Message;
END_VAR

  _stMsg.eType               := E_MessageType.eMessageInfo;
  _stMsg.eDevice             := E_Device.NciChannelCtrl + TO_UINT(ChnId);
  _stMsg.eSubdevice          := e_Subdevice.NciControl;
  _stMsg.iErrorNumber        := 0;

  _sCtrl                     := concat('E_NCI_CTRL', '.');
  _sCtrl                     := concat(_sCtrl, TO_STRING(_eCtrlOld));

  _sResult                   := concat(': E_PROGRESS', '.');
  _sResult                   := concat(_sResult, TO_STRING(_eResult));

  _stMsg.sText               := concat(_sCtrl, ' ');
  _stMsg.sText               := concat(_sCtrl, _sResult);

  IF (_MessageLevel < E_MessageType.eMessageError)
  THEN
    f_MessageSet(_stMsg);
  ELSE
    IF (_stMsg.eType = E_MessageType.eMessageError)
    THEN
      f_MessageSet(_stMsg);
    END_IF
  END_IF
END_METHOD

PROPERTY M_FunctionScope : pointer to st_nci_m_func
SET
_MFuncScope := M_FunctionScope;
END_SET
END_PROPERTY

END_FUNCTION_BLOCK

// ---- APPLICATION/_types/LinkedList/fb_Process_LinkedList.TcPOU
//---------------------------------------------------------------------------------------------------------------
//
//  HAUD 2025.02.24
//
//  - fb_LinkedList
//  -----------------------------
//  - library wrapper for linked list
//---------------------------------------------------------------------------------------------------------------
FUNCTION_BLOCK fb_Process_LinkedList IMPLEMENTS I_Process_LinkedList
VAR
  _LastNodeAdded,
  _LastNodeRemoved  : ST_PROCESS_LIST_RESULT;

	_nCount           : UDINT;
  _nFree            : UDINT;

  {attribute 'hide'}
	_stList           : ARRAY[0..MAX_LIST_NODES] OF ST_PROCESS_DATA;
	_stNodes          : ARRAY[0..MAX_LIST_NODES] OF T_LinkedListEntry;

	_fbList           : Tc2_Utilities.FB_LinkedListCtrl;
	_hList            : Tc2_Utilities.T_HLINKEDLIST;

	_stRef            : POINTER TO ST_PROCESS_DATA;
END_VAR

METHOD AddHeadValue : ST_PROCESS_LIST_RESULT
VAR_INPUT
  stData        : ST_PROCESS_DATA;
END_VAR
VAR
  _nIdxNode     : ULINT; 
	_pPosGet      : POINTER TO T_LinkedListEntry;
  _stRes        : ST_PROCESS_LIST_RESULT;
END_VAR

// add empty node
_fbList.A_AddHeadValue( hList     := _hList, 
                        putValue  := 16#0, 
                        getPosPtr => _pPosGet);

IF NOT _fbList.bOk 
THEN
  _stRes.wState.0       := TRUE;
ELSE
  // Get array index of new node
	_fbList.A_GetIndexAtPosPtr( hList       := _hList, 
                              putPosPtr   := _pPosGet, 
                              getValue    => _nIdxNode);

	IF NOT _fbList.bOk 
  THEN
    _stRes.wState.1     := TRUE;
  ELSE
    // write data to new node index
		_stRef 	            := ADR( _stList[_nIdxNode] );
		_stRef^ 	          := stData;

		_fbList.A_SetValueAtPosPtr( hList     := _hList, 
                                putPosPtr := _pPosGet, 
                                putValue  := _stRef);

		IF NOT _fbList.bOk 
    THEN
      _stRes.wState.2   := TRUE;
    ELSE
      _stRes.nIndex     := _nIdxNode;
			_stRes.stData     := stData;
      _LastNodeAdded    := _stRes;
		END_IF
	END_IF
END_IF
_nCount                 := _hList.nCount;
_nFree                  := _hList.nFree;
AddHeadValue            := _stRes;
END_METHOD

METHOD AddTailValue : ST_PROCESS_LIST_RESULT
VAR_INPUT
  stData        : ST_PROCESS_DATA;
END_VAR
VAR
  _nIdxNode     : ULINT; 
	_pPosGet      : POINTER TO T_LinkedListEntry;
  _stRes        : ST_PROCESS_LIST_RESULT;
END_VAR

// add empty node
_fbList.A_AddTailValue( hList       := _hList, 
                        putValue    := 16#0, 
                        getPosPtr   => _pPosGet);


IF NOT _fbList.bOk 
THEN
  _stRes.wState.0       := TRUE;
ELSE
  // Get array index of new node
	_fbList.A_GetIndexAtPosPtr( hList       := _hList, 
                              putPosPtr   := _pPosGet, 
                              getValue    => _nIdxNode);

	IF NOT _fbList.bOk 
  THEN
    _stRes.wState.1     := TRUE;
  ELSE
    // write data to new node index
		_stRef 	            := ADR( _stList[_nIdxNode] );
		_stRef^ 	          := stData;

		_fbList.A_SetValueAtPosPtr( hList     := _hList, 
                                putPosPtr := _pPosGet, 
                                putValue  := _stRef);

		IF NOT _fbList.bOk 
    THEN
      _stRes.wState.2   := TRUE;
    ELSE
      _stRes.nIndex     := _nIdxNode;
			_stRes.stData     := stData;
      _LastNodeAdded    := _stRes;
		END_IF
	END_IF
END_IF
_nCount                 := _hList.nCount;
_nFree                  := _hList.nFree;
AddTailValue            := _stRes;
END_METHOD

PROPERTY Count : UDINT
GET
Count := _nCount := _hList.nCount;
END_GET
END_PROPERTY

PROPERTY Data : ARRAY[1..MAX_LIST_NODES] OF ST_PROCESS_DATA
GET
VAR
	_tList        : ARRAY[1..MAX_LIST_NODES] OF ST_PROCESS_DATA;
  _getValue     : PVOID;
  _pEntry       : POINTER TO ST_PROCESS_DATA;
  _getPosPtr    : POINTER TO T_LinkedListEntry := 0;
  _nIdx         : UINT;  
END_VAR
_fbList(
	hList       := _hList);

_nCount       := _hList.nCount;
_nFree        := _hList.nFree;


_fbList.A_GetHead( hList := _hList, getValue=> _getValue, getPosPtr=> _getPosPtr );
IF _fbList.bOk 
THEN
  IF (_hList.nCount > 0)
  THEN
    _nIdx         := 1;
    _pEntry       := _getValue;
    _tList[1]     := _pEntry^;
    
    REPEAT
      _fbList.A_GetNext( hList := _hList, putPosPtr := _getPosPtr, getValue=> _getValue, getPosPtr=> _getPosPtr );
  
      IF _fbList.bOk THEN
        _nIdx         := _nIdx + 1;
        _pEntry       := _getValue;
        _tList[_nIdx] := _pEntry^;
      ELSE
        EXIT;
      END_IF
    UNTIL NOT _fbList.bOk
    END_REPEAT
  END_IF
END_IF

Data := _tList;
END_GET
END_PROPERTY

PROPERTY Free : UDINT
GET
Free := _nFree := _hList.nFree;
END_GET
END_PROPERTY

METHOD GetHead : ST_PROCESS_LIST_RESULT
VAR_INPUT
END_VAR
VAR
	_pPosGet      : POINTER TO T_LinkedListEntry;
  _pData        : POINTER TO ST_PROCESS_DATA;
  _stRes        : ST_PROCESS_LIST_RESULT;
END_VAR

_fbList.A_GetHead(  hList      := _hList,
                    getValue   => _pData,
                    getPosPtr  => _pPosGet);

IF NOT _fbList.bOk
THEN
  _stRes.wState.0   := TRUE;
ELSE
  _stRes.stData     := _pData^;
END_IF
_nCount             := _hList.nCount;
_nFree              := _hList.nFree;
GetHead             := _stRes;
END_METHOD

METHOD GetTail : ST_PROCESS_LIST_RESULT
VAR_INPUT
END_VAR
VAR
	_pPosGet      : POINTER TO T_LinkedListEntry;
  _pData        : POINTER TO ST_PROCESS_DATA;
  _stRes        : ST_PROCESS_LIST_RESULT;
END_VAR

_fbList.A_GetTail(  hList      := _hList,
                    getValue   => _pData,
                    getPosPtr  => _pPosGet);

IF NOT _fbList.bOk
THEN
  _stRes.wState.0   := TRUE;
ELSE
  _stRes.stData     := _pData^;
END_IF
_nCount             := _hList.nCount;
_nFree              := _hList.nFree;
GetTail             := _stRes;
END_METHOD

METHOD InitList : BOOL
VAR_INST
  _bOk        : BOOL;
  _bListinit  : BOOL;
END_VAR
                         // Tc2_Utilities
_bListInit            := F_CreateLinkedListHnd(
                              ADR   (_stNodes), 
                              SIZEOF(_stNodes), 
                              _hList          );

IF _bListInit
THEN
  _fbList.A_Reset(hList   := _hList, 
                  bOk     => _bOk);

  memset(ADR(_stList), 0, SIZEOF(_stList));

  _nCount                 := _hList.nCount;
  _nFree                  := _hList.nFree;
  InitList                := TRUE; //_bOk;
END_IF
END_METHOD

PROPERTY Nodes : ARRAY[0..MAX_LIST_NODES] OF T_LinkedListEntry
GET
Nodes := _stNodes;
END_GET
END_PROPERTY

METHOD RemoveHeadValue : ST_PROCESS_LIST_RESULT
VAR_INPUT
END_VAR
VAR
	_pPosGet      : POINTER TO T_LinkedListEntry;
  _pData        : POINTER TO ST_PROCESS_DATA;
  _stRes        : ST_PROCESS_LIST_RESULT;
END_VAR
_fbList.A_RemoveHeadValue(hList       := _hList, 
                          getValue    => _pData, 
                          getPosPtr   => _pPosGet);

IF NOT _fbList.bOk 
THEN
  _stRes.wState.0   := TRUE;
ELSE
	_stRes.stData     := _pData^;
  _LastNodeRemoved  := _stRes;

  memset(_pData, 0, SIZEOF(ST_PROCESS_DATA));
END_IF
_nCount             := _hList.nCount;
_nFree              := _hList.nFree;
RemoveHeadValue     := _stRes;
END_METHOD

METHOD RemoveTailValue : ST_PROCESS_LIST_RESULT
VAR_INPUT
END_VAR
VAR
	_pPosGet      : POINTER TO T_LinkedListEntry;
  _pData        : POINTER TO ST_PROCESS_DATA;
  _stRes        : ST_PROCESS_LIST_RESULT;
END_VAR
_fbList.A_RemoveTailValue(hList       := _hList, 
                          getValue    => _pData, 
                          getPosPtr   => _pPosGet);

IF NOT _fbList.bOk 
THEN
  _stRes.wState.0   := TRUE;
ELSE
	_stRes.stData     := _pData^;
  _LastNodeRemoved  := _stRes;

  memset(_pData, 0, SIZEOF(ST_PROCESS_DATA));
END_IF
_nCount             := _hList.nCount;
_nFree              := _hList.nFree;
RemoveTailValue     := _stRes;
END_METHOD

END_FUNCTION_BLOCK

// ---- PLC_MOTION/CAM/class/FB_CamAxis.TcPOU
FUNCTION_BLOCK abstract FB_CamAxis
VAR
  _eCheck                       : E_CHECK_STATE;
  _nErrorId                     : UDINT; // datafield for error

  _MessageLevel                 : E_MessageType;

  _AxisSlave                    : REFERENCE TO AXIS_REF;
  _AxisMaster                   : REFERENCE TO AXIS_REF;

  _fbCamInV2                    : Tc2_MC2_Camming.MC_CamIn_V2;
  _fbScalingV2                  : Tc2_MC2_Camming.MC_CamScaling_V2;
  _fbCamInfoV2                  : Tc2_MC2_Camming.MC_CamInfo_V2;

  _fbCamOut                     : Tc2_MC2_Camming.MC_CamOut;

  _fbSetCamOnlineChangeMode     : Tc2_MC2_Camming.MC_SetCamOnlineChangeMode;

  _fbReadMotionFunction         : Tc2_MC2_Camming.MC_ReadMotionFunction;
  _fbReadMotionFunctionPoint    : Tc2_MC2_Camming.MC_ReadMotionFunctionPoint;
  _fbReadMotionFunctionValues   : Tc2_MC2_Camming.MC_ReadMotionFunctionValues;

  _fbWriteMotionFunction        : Tc2_MC2_Camming.MC_WriteMotionFunction;
  _fbWriteMotionFunctionPoint   : Tc2_MC2_Camming.MC_WriteMotionFunctionPoint;

  _stCamData                    : ST_CAM_DATA;  // camming parameters for function calls

  _mcCamInfoData                : Tc2_MC2_Camming.MC_CamInfoData; // read cam info from NC

  _mcCamRef                     : MC_CAM_REF;
  _mcMotionFunction             : ARRAY[1..MAX_MOTION_FUNCTION_POINTS] OF Tc2_MC2_Camming.MC_MotionFunctionPoint;
  _mcMotionFunctionPoint        : Tc2_MC2_Camming.MC_MotionFunctionPoint;
  _nMotionFunctionSize          : UINT;
END_VAR

METHOD CamIn : E_PROGRESS
VAR_INPUT
  Execute           : BOOL;
  nMasterIndex      : UINT;
END_VAR
VAR_INST
  _eCk              : E_CHECK_STATE;
  _eState           : E_PROGRESS;
  _rValue           : LREAL;
  _udiErr           : UDINT;
  _stMsg            : ST_Message;
END_VAR
IF NOT __ISVALIDREF(_AxisSlave)
THEN
  _eCheck                     := E_CHECK_STATE.CAM_SLAVE_AXIS_REF_INVALID;
  CamIn                       := E_PROGRESS.PROGRESS_ERROR;
  RETURN;
END_IF

IF NOT Execute THEN _eState := E_PROGRESS.PROGRESS_INIT; END_IF


CASE _eState
OF
  E_PROGRESS.PROGRESS_INIT:
    IF Execute 
    THEN
      memset(ADR(_stMsg),0,SIZEOF(_stMsg));
      _udiErr                       := 0;

      IF NOT (nMasterIndex = _stCamData.nMasterIndex)
      THEN
        _eState                     := E_PROGRESS.PROGRESS_ERROR;
        _eCk                        := E_CHECK_STATE.CAM_MASTER_AXIS_REF_INVALID;

        _stMsg.eType                := E_MessageType.eMessageError;
        _stMsg.eDevice              := E_Device.Camming + (_AxisSlave.NcToPlc.AxisId);
        _stMsg.eSubdevice           := e_Subdevice.fbCamInV2;
        _stMsg.iErrorNumber         := nMasterIndex;
  
        _stMsg.sText                := concat(' : ', TO_STRING(_eCk));
        f_MessageSet(_stMsg);

      ELSE
        _eState                     := E_PROGRESS.PROGRESS_BUSY;
        _eCk                        := E_CHECK_STATE.CHECK_DONE;

        IF (_MessageLevel = E_MessageType.eMessageVerbose)
        THEN
          _stMsg.eType              := E_MessageType.eMessageVerbose;
          _stMsg.eDevice            := E_Device.Camming + (_AxisSlave.NcToPlc.AxisId);
          _stMsg.eSubdevice         := e_Subdevice.fbCamInfoV2;
          _stMsg.iErrorNumber       := 0;
    
          _stMsg.sText              := concat(' : ', TO_STRING(_eState));
          f_MessageSet(_stMsg);
        END_IF

      _fbCamInV2(
          Master                    := _AxisMaster, 
          Slave                     := _AxisSlave, 
          Execute                   := FALSE, 
          ActivationMode            := _stCamData.nActivationMode, 
          ActivationPosition        := _stCamData.rActivationPosition, 
          CamTableID                := _stCamData.nCamTableId,
          Scaling                   := CamScalingData,
          Options                   := CamInOptions);
      END_IF
    END_IF
END_CASE
CASE _eState
OF
  E_PROGRESS.PROGRESS_BUSY:
    _fbCamInV2(
          Master                    := _AxisMaster, 
          Slave                     := _AxisSlave, 
          Execute                   := TRUE, 
          ActivationMode            := _stCamData.nActivationMode, 
          ActivationPosition        := _stCamData.rActivationPosition, 
          CamTableID                := _stCamData.nCamTableId);

    IF (_fbCamInV2.Error)
    THEN
      _eState                       := E_PROGRESS.PROGRESS_ERROR;
      _udiErr                       := _fbCamInV2.ErrorID;

      _stMsg.eType                  := E_MessageType.eMessageError;
      _stMsg.eDevice                := E_Device.Camming + (_AxisSlave.NcToPlc.AxisId);
      _stMsg.eSubdevice             := e_Subdevice.fbCamInV2;
      _stMsg.iErrorNumber           := _udiErr;

      _stMsg.sText                  := concat(' : ', TO_STRING(_eState));
      f_MessageSet(_stMsg);

      _fbCamInV2(
          Master                    := _AxisMaster, 
          Slave                     := _AxisSlave, 
          Execute                   := FALSE); 

    ELSIF (_fbCamInV2.InSync)
    THEN
      _eState                       := E_PROGRESS.PROGRESS_DONE;

      IF (_MessageLevel > E_MessageType.eMessageError)
      THEN
        _stMsg.eType                := E_MessageType.eMessageInfo;
        _stMsg.eDevice              := E_Device.Camming + (_AxisSlave.NcToPlc.AxisId);
        _stMsg.eSubdevice           := e_Subdevice.fbCamInV2;
        _stMsg.iErrorNumber         := 0;
  
        _stMsg.sText                := concat(' : ', TO_STRING(_eState));
        f_MessageSet(_stMsg);
      END_IF

      _fbCamInV2(
          Master                    := _AxisMaster, 
          Slave                     := _AxisSlave, 
          Execute                   := FALSE); 
    END_IF
END_CASE

CamIn                               := _eState;
END_METHOD

METHOD CamInfo : E_PROGRESS
VAR_INPUT
  Execute           : BOOL;
  CamTableID        : Tc2_MC2_Camming.MC_CAM_ID;
  AtMasterPosition  : BOOL;
  MasterPosition    : LREAL;
END_VAR
VAR_INST
  _eState           : E_PROGRESS;
  _rValue           : LREAL;
  _udiErr           : UDINT;
  _stMsg            : ST_Message;
  _stCID            : Tc2_MC2_Camming.MC_CamInfoData;
END_VAR

IF NOT __ISVALIDREF(_AxisSlave)
THEN
  _eCheck                     := E_CHECK_STATE.CAM_SLAVE_AXIS_REF_INVALID;
  CamInfo                     := E_PROGRESS.PROGRESS_ERROR;
  RETURN;
END_IF

IF NOT Execute THEN _eState := E_PROGRESS.PROGRESS_INIT; END_IF

CASE _eState
OF
  E_PROGRESS.PROGRESS_INIT:
    IF Execute 
    THEN
      memset(ADR(_stMsg),0,SIZEOF(_stMsg));
      memset(ADR(_stCID),0,SIZEOF(_stCID));

      _udiErr                       := 0;
      _eState                       := E_PROGRESS.PROGRESS_BUSY;

      _fbCamInfoV2(
              Slave                 := _AxisSlave, 
              Execute               := FALSE, 
              CamTableID            := CamTableID, 
              AtMasterPosition      := AtMasterPosition, 
              MasterPosition        := MasterPosition,
              CamInfo               => _mcCamInfoData);

      IF (_MessageLevel = E_MessageType.eMessageVerbose)
      THEN
        _stMsg.eType                := E_MessageType.eMessageVerbose;
        _stMsg.eDevice              := E_Device.Camming + (_AxisSlave.NcToPlc.AxisId);
        _stMsg.eSubdevice           := e_Subdevice.fbCamInfoV2;
        _stMsg.iErrorNumber         := 0;
  
        _stMsg.sText                := concat(' : ', TO_STRING(_eState));
        f_MessageSet(_stMsg);
      END_IF
    END_IF
END_CASE
CASE _eState
OF
  E_PROGRESS.PROGRESS_BUSY:
    _fbCamInfoV2(
              Slave                 := _AxisSlave, 
              Execute               := TRUE, 
              CamTableID            := CamTableID, 
              AtMasterPosition      := AtMasterPosition, 
              MasterPosition        := MasterPosition,
              CamInfo               => _mcCamInfoData);

    IF (_fbCamInfoV2.Error)
    THEN
      _eState                       := E_PROGRESS.PROGRESS_ERROR;
      _udiErr                       := _fbCamInfoV2.ErrorID;

      _stMsg.eType                  := E_MessageType.eMessageError;
      _stMsg.eDevice                := E_Device.Camming + (_AxisSlave.NcToPlc.AxisId);
      _stMsg.eSubdevice             := e_Subdevice.fbCamInfoV2;
      _stMsg.iErrorNumber           := _udiErr;

      _stMsg.sText                  := concat(' : ', TO_STRING(_eState));
      f_MessageSet(_stMsg);

      _fbCamInfoV2(
              Slave                 := _AxisSlave, 
              Execute               := FALSE);

    ELSIF (_fbCamInfoV2.Done)
    THEN
      _eState                       := E_PROGRESS.PROGRESS_DONE;
      _stCID                        := _fbCamInfoV2.CamInfo;

      IF (_MessageLevel > E_MessageType.eMessageError)
      THEN
        _stMsg.eType                := E_MessageType.eMessageInfo;
        _stMsg.eDevice              := E_Device.Camming + (_AxisSlave.NcToPlc.AxisId);
        _stMsg.eSubdevice           := e_Subdevice.fbCamInfoV2;
        _stMsg.iErrorNumber         := 0;
  
        _stMsg.sText                := concat(' : ', TO_STRING(_eState));
        f_MessageSet(_stMsg);
      END_IF
      _fbCamInfoV2(
              Slave                 := _AxisSlave, 
              Execute               := FALSE);
    END_IF
END_CASE

CamInfo                             := _eState;
END_METHOD

PROPERTY CamInfoData : ST_CAM_INFO
GET
VAR
  _stInfoData     : ST_CAM_INFO;
END_VAR


_stInfoData.bPeriodic                       := _mcCamInfoData.Periodic;
_stInfoData.bMasterAbsolute                 := _mcCamInfoData.MasterAbsolute;
_stInfoData.bSlaveAbsolute                  := _mcCamInfoData.SlaveAbsolute;
_stInfoData.bScalingPending                 := _mcCamInfoData.ScalingPending;
_stInfoData.bCamDataQueued                  := _mcCamInfoData.CamDataQueued;
_stInfoData.bCamTableQueued                 := _mcCamInfoData.CamTableQueued;

_stInfoData.nTableType                      := _mcCamInfoData.TableType;
_stInfoData.nInterpolationType              := _mcCamInfoData.InterpolationType;
_stInfoData.nNumberOfRows                   := TO_UINT(_mcCamInfoData.NumberOfRows);
_stInfoData.nNumberOfColumns                := TO_UINT(_mcCamInfoData.NumberOfColumns);
_stInfoData.nMasterAxisId                   := TO_UINT(_mcCamInfoData.MasterAxisId);
_stInfoData.nSlaveAxisId                    := TO_UINT(_mcCamInfoData.SlaveAxisId);

_stInfoData.rMasterCamStartPos              := _mcCamInfoData.MasterCamStartPos;
_stInfoData.rSlaveCamStartPos               := _mcCamInfoData.SlaveCamStartPos;
_stInfoData.rRawMasterPeriod                := _mcCamInfoData.RawMasterPeriod;
_stInfoData.rRawSlaveStroke                 := _mcCamInfoData.RawSlaveStroke;
_stInfoData.rMasterAxisCouplingPos          := _mcCamInfoData.MasterAxisCouplingPos;
_stInfoData.rSlaveAxisCouplingPos           := _mcCamInfoData.SlaveAxisCouplingPos;

_stInfoData.rMasterOffset                   := _mcCamInfoData.MasterOffset;
_stInfoData.rSlaveOffset                    := _mcCamInfoData.SlaveOffset;
_stInfoData.rMasterScaling                  := _mcCamInfoData.MasterScaling;
_stInfoData.rSlaveScaling                   := _mcCamInfoData.SlaveScaling;
_stInfoData.rSumOfSlaveStrokes              := _mcCamInfoData.SumOfSlaveStrokes;
_stInfoData.rSumOfSuperpositionDistance     := _mcCamInfoData.SumOfSuperpositionDistance;
_stInfoData.rActualMasterAxisPos            := _mcCamInfoData.ActualMasterAxisPos;
_stInfoData.rActualSlaveAxisPos             := _mcCamInfoData.ActualSlaveAxisPos;
_stInfoData.rActualMasterCamPos             := _mcCamInfoData.ActualMasterCamPos;
_stInfoData.rActualSlaveCamPos              := _mcCamInfoData.ActualSlaveCamPos;
_stInfoData.rActualPhaseShift               := _mcCamInfoData.ActualPhaseShift;

_stInfoData.nScalingActivationMode          := _mcCamInfoData.ScalingActivationMode;
_stInfoData.rScalingActivationPos           := _mcCamInfoData.ScalingActivationPos;
_stInfoData.nScalingMasterScalingMode       := _mcCamInfoData.ScalingMasterScalingMode;
_stInfoData.nScalingSlaveScalingMode        := _mcCamInfoData.ScalingSlaveScalingMode;

_stInfoData.nOnlineChangeActivationMode     := _mcCamInfoData.OnlineChangeActivationMode;
_stInfoData.rOnlineChangeActivationPos      := _mcCamInfoData.OnlineChangeActivationPos;
_stInfoData.nOnlineChangeMasterScalingMode  := _mcCamInfoData.OnlineChangeMasterScalingMode;
_stInfoData.nOnlineChangeSlaveScalingMode   := _mcCamInfoData.OnlineChangeSlaveScalingMode;

_stInfoData.nCamExchangeCamTableID          := _mcCamInfoData.CamExchangeCamTableID;
_stInfoData.nCamExchangeActivationMode      := _mcCamInfoData.CamExchangeActivationMode;
_stInfoData.rCamExchangeActivationPos       := _mcCamInfoData.CamExchangeActivationPos;
_stInfoData.nCamExchangeMasterScalingMode   := _mcCamInfoData.CamExchangeMasterScalingMode;
_stInfoData.nCamExchangeSlaveScalingMode    := _mcCamInfoData.CamExchangeSlaveScalingMode;
END_GET
END_PROPERTY

PROPERTY CamInOptions : ST_CamInOptions_V2
GET
VAR
  _CamInOptions   : ST_CamInOptions_V2;
END_VAR

_CamInOptions.CamOperationMode      := _stCamData.stOptions.nCamOperationMode;
_CamInOptions.InterpolationType     := _stCamData.stOptions.nInterpolationType;
_CamInOptions.ReferenceCamTableID   := _stCamData.stOptions.nReferenceCamTableId;
END_GET
END_PROPERTY

METHOD CamOut : E_PROGRESS
VAR_INPUT
  Execute           : BOOL;
END_VAR
VAR_INST
  _dwCoupleState    : DWORD;      // debug
  _eState           : E_PROGRESS;
  _rValue           : LREAL;
  _udiErr           : UDINT;
  _stMsg            : ST_Message;
END_VAR

IF NOT __ISVALIDREF(_AxisSlave)
THEN
  _eCheck                     := E_CHECK_STATE.CAM_SLAVE_AXIS_REF_INVALID;
  CamOut                      := E_PROGRESS.PROGRESS_ERROR;
  RETURN;
END_IF

IF NOT Execute THEN _eState := E_PROGRESS.PROGRESS_INIT; END_IF


CASE _eState
OF
  E_PROGRESS.PROGRESS_INIT:
    IF Execute 
    THEN
      memset(ADR(_stMsg),0,SIZEOF(_stMsg));
      _udiErr                       := 0;
      _dwCoupleState                := _AxisSlave.NcToPlc.CoupleState;

      _eState                       := E_PROGRESS.PROGRESS_BUSY;

      IF (_MessageLevel = E_MessageType.eMessageVerbose)
      THEN
        _stMsg.eType                := E_MessageType.eMessageInfo;
        _stMsg.eDevice              := E_Device.Camming + (_AxisSlave.NcToPlc.AxisId);
        _stMsg.eSubdevice           := e_Subdevice.fbCamOut;
        _stMsg.iErrorNumber         := 0;
  
        _stMsg.sText                := concat(' : ', TO_STRING(_eState));
        f_MessageSet(_stMsg);
      END_IF
      _fbCamOut(
                Slave               := _AxisSlave, 
                Execute             := FALSE);
    END_IF
END_CASE
CASE _eState
OF
  E_PROGRESS.PROGRESS_BUSY:
    _fbCamOut(
              Slave                 := _AxisSlave, 
              Execute               := TRUE);

    IF (_fbCamOut.Error)
    THEN
      _eState                       := E_PROGRESS.PROGRESS_ERROR;
      _udiErr                       := _fbCamOut.ErrorID;

      _stMsg.eType                  := E_MessageType.eMessageError;
      _stMsg.eDevice                := E_Device.Camming + (_AxisSlave.NcToPlc.AxisId);
      _stMsg.eSubdevice             := e_Subdevice.fbCamOut;
      _stMsg.iErrorNumber           := _udiErr;

      _stMsg.sText                  := concat(' : ', TO_STRING(_eState));
      f_MessageSet(_stMsg);

      _fbCamOut(
                Slave               := _AxisSlave, 
                Execute             := FALSE);

    ELSIF (_fbCamOut.Done)
    THEN
      _eState                       := E_PROGRESS.PROGRESS_DONE;

      IF (_MessageLevel > E_MessageType.eMessageError)
      THEN
        _stMsg.eType                := E_MessageType.eMessageInfo;
        _stMsg.eDevice              := E_Device.Camming + (_AxisSlave.NcToPlc.AxisId);
        _stMsg.eSubdevice           := e_Subdevice.fbCamOut;
        _stMsg.iErrorNumber         := 0;
  
        _stMsg.sText                := concat(' : ', TO_STRING(_eState));
        f_MessageSet(_stMsg);
      END_IF
      _fbCamOut(
                Slave               := _AxisSlave, 
                Execute             := FALSE);
    END_IF
END_CASE

CamOut                              := _eState;
END_METHOD

METHOD CamScaling : E_PROGRESS
VAR_INPUT
  Execute           : BOOL;
END_VAR
VAR_INST
  _eState           : E_PROGRESS;
  _rValue           : LREAL;
  _udiErr           : UDINT;
  _stMsg            : ST_Message;

  _stLastScalingData  : Tc2_MC2_Camming.ST_CamScalingData;
  _nLastCamTableID    : UDINT;
END_VAR
IF NOT __ISVALIDREF(_AxisSlave)
THEN
  _eCheck                     := E_CHECK_STATE.CAM_SLAVE_AXIS_REF_INVALID;
  CamScaling                  := E_PROGRESS.PROGRESS_ERROR;
  RETURN;
END_IF

IF NOT Execute THEN _eState   := E_PROGRESS.PROGRESS_INIT; END_IF


CASE _eState
OF
  E_PROGRESS.PROGRESS_INIT:
    IF Execute 
    THEN
      memset(ADR(_stMsg),0,SIZEOF(_stMsg));
      _udiErr                       := 0;
      _rValue                       := 0;
      _eState                       := E_PROGRESS.PROGRESS_BUSY;

      _fbScalingV2(
              Slave                 := _AxisSlave, 
              Execute               := FALSE, 
              ActivationMode        := _stCamData.nActivationMode, 
              ActivationPosition    := _stCamData.rActivationPosition, 
              CamTableID            := _stCamData.nCamTableId,
              Scaling               := CamScalingData);
    END_IF
END_CASE
CASE _eState
OF
  E_PROGRESS.PROGRESS_BUSY:
    _eState                         := E_PROGRESS.PROGRESS_STARTUP;
    _nLastCamTableID                := _stCamData.nCamTableId;
    _stLastScalingData              := _fbScalingV2.Scaling;

    IF (_MessageLevel = E_MessageType.eMessageVerbose)
    THEN
      _stMsg.eType                  := E_MessageType.eMessageVerbose;
      _stMsg.eDevice                := E_Device.Camming + (_AxisSlave.NcToPlc.AxisId);
      _stMsg.eSubdevice             := e_Subdevice.fbCamScalingV2;
      _stMsg.iErrorNumber           := _nLastCamTableID;

      _stMsg.sText                  := concat(' : ', TO_STRING(_eState));
      f_MessageSet(_stMsg);
    END_IF
END_CASE
CASE _eState
OF
  E_PROGRESS.PROGRESS_STARTUP:
      _fbScalingV2(
              Slave                 := _AxisSlave, 
              Execute               := TRUE, 
              ActivationMode        := _stCamData.nActivationMode, 
              ActivationPosition    := _stCamData.rActivationPosition, 
              CamTableID            := _stCamData.nCamTableId);

    IF (_fbScalingV2.Error)
    THEN
      _eState                       := E_PROGRESS.PROGRESS_ERROR;
      _udiErr                       := _fbScalingV2.ErrorID;

      _stMsg.eType                  := E_MessageType.eMessageError;
      _stMsg.eDevice                := E_Device.Camming + (_AxisSlave.NcToPlc.AxisId);
      _stMsg.eSubdevice             := e_Subdevice.fbCamScalingV2;
      _stMsg.iErrorNumber           := _udiErr;

      _stMsg.sText                  := concat(' : ', TO_STRING(_eState));
      f_MessageSet(_stMsg);

      _fbScalingV2(
              Slave                 := _AxisSlave, 
              Execute               := FALSE); 

    ELSIF (_fbScalingV2.CommandAborted)
    THEN
      _eState                       := E_PROGRESS.PROGRESS_ERROR;
      _udiErr                       := _fbScalingV2.ErrorID;

      _stMsg.eType                  := E_MessageType.eMessageError;
      _stMsg.eDevice                := E_Device.Camming + (_AxisSlave.NcToPlc.AxisId);
      _stMsg.eSubdevice             := e_Subdevice.fbCamScalingV2;
      _stMsg.iErrorNumber           := _udiErr;

      _stMsg.sText                  := concat('command aborted : ', TO_STRING(_eState));
      f_MessageSet(_stMsg);

      _fbScalingV2(
          Slave                     := _AxisSlave, 
          Execute                   := FALSE); 

    ELSIF (_fbScalingV2.Done)
    THEN
      _eState                       := E_PROGRESS.PROGRESS_DONE;

      IF (_MessageLevel > E_MessageType.eMessageError)
      THEN
        _stMsg.eType                := E_MessageType.eMessageInfo;
        _stMsg.eDevice              := E_Device.Camming + (_AxisSlave.NcToPlc.AxisId);
        _stMsg.eSubdevice           := e_Subdevice.fbCamScalingV2;
        _stMsg.iErrorNumber         := 0;
  
        _stMsg.sText                := concat(' : ', TO_STRING(_eState));
        f_MessageSet(_stMsg);
      END_IF
      _fbScalingV2(
              Slave                 := _AxisSlave, 
              Execute               := FALSE); 
    END_IF
END_CASE

CamScaling                          := _eState;
END_METHOD

PROPERTY CamScalingData : Tc2_MC2_Camming.ST_CamScalingData
GET
VAR
 _ScaleData   : Tc2_MC2_Camming.ST_CamScalingData;
END_VAR

_ScaleData.MasterOffset       := _stCamData.stCamScalingData.rMasterOffset;
_ScaleData.MasterRelative     := _stCamData.stCamScalingData.bMasterRelative;
_ScaleData.MasterScaling      := _stCamData.stCamScalingData.rMasterScaling;
_ScaleData.MasterScalingMode  := _stCamData.stCamScalingData.nMasterScalingMode;

_ScaleData.SlaveOffset        := _stCamData.stCamScalingData.rSlaveOffset;
_ScaleData.SlaveRelative      := _stCamData.stCamScalingData.bSlaveRelative;
_ScaleData.SlaveScaling       := _stCamData.stCamScalingData.rSlaveScaling;
_ScaleData.SlaveScalingMode   := _stCamData.stCamScalingData.nSlaveScalingMode;

CamScalingData                := _ScaleData;
END_GET
END_PROPERTY

PROPERTY MessageLevel : E_MessageType
SET
_MessageLevel := MessageLevel;
END_SET
END_PROPERTY

METHOD ReadMotionFunction : E_PROGRESS
VAR_INPUT
  Execute           : BOOL;
END_VAR
VAR_INST
  _eState           : E_PROGRESS;
  _rValue           : LREAL;
  _udiErr           : UDINT;
  _stMsg            : ST_Message;


  _nNumPointsRead   : UINT;
END_VAR
IF NOT Execute THEN _eState   := E_PROGRESS.PROGRESS_INIT; END_IF


CASE _eState
OF
  E_PROGRESS.PROGRESS_INIT:
    IF Execute 
    THEN
      memset(ADR(_mcMotionFunction),0,SIZEOF(_mcMotionFunction));
      memset(ADR(_stMsg),0,SIZEOF(_stMsg));
      _nNumPointsRead               := 0;
      _udiErr                       := 0;
      _rValue                       := 0;
      _eState                       := E_PROGRESS.PROGRESS_BUSY;

      _mcCamRef.pArray              := ADR(_mcMotionFunction);
      _mcCamRef.ArraySize           := SIZEOF(_mcMotionFunction);

      _mcCamRef.TableType           := Tc2_MC2_Camming.MC_TABLETYPE_MOTIONFUNCTION;
      _mcCamRef.NoOfColumns         := 1;

      _fbReadMotionFunction(
              Execute               := FALSE, 
              CamTableID            := _stCamData.nCamTableId, 
              PointID               := _stCamData.nPointId,     // must be greater 0
              NumPoints             := _stCamData.nNumPoints,   // 0 = read all
              CamTable              := _mcCamRef);

    END_IF
END_CASE
CASE _eState
OF
  E_PROGRESS.PROGRESS_BUSY:
    _fbReadMotionFunction(
              Execute               := TRUE, 
              CamTableID            := _stCamData.nCamTableId,  // ID of the loaded table
              PointID               := _stCamData.nPointId,     // Point ID of the first point to be read
              NumPoints             := _stCamData.nNumPoints,   // 0 = read all points
              CamTable              := _mcCamRef);

    IF (_fbReadMotionFunction.Error)
    THEN
      _eState                       := E_PROGRESS.PROGRESS_ERROR;
      _udiErr                       := _fbReadMotionFunction.ErrorID;

      _stMsg.eType                  := E_MessageType.eMessageError;
      _stMsg.eDevice                := E_Device.Camming + (_AxisSlave.NcToPlc.AxisId);
      _stMsg.eSubdevice             := e_Subdevice.fbReadMotionFunction;
      _stMsg.iErrorNumber           := _udiErr;

      _stMsg.sText                  := concat(' : ', TO_STRING(_eState));
      f_MessageSet(_stMsg);

      _fbReadMotionFunction(
              Execute               := FALSE, 
              CamTableID            := _stCamData.nCamTableId,  // ID of the loaded table
              PointID               := _stCamData.nPointId,     // Point ID of the first point to be read
              NumPoints             := _stCamData.nNumPoints,   // 0 = read all points
              CamTable              := _mcCamRef);

    ELSIF (_fbReadMotionFunction.Done)
    THEN
      _eState                       := E_PROGRESS.PROGRESS_WORKING;

      IF (_MessageLevel < E_MessageType.eMessageError)
      THEN
        _stMsg.eType                := E_MessageType.eMessageInfo;
        _stMsg.eDevice              := E_Device.Camming + (_AxisSlave.NcToPlc.AxisId);
        _stMsg.eSubdevice           := e_Subdevice.fbReadMotionFunction;
        _stMsg.iErrorNumber         := 0;
  
        _stMsg.sText                := concat(' : ', TO_STRING(_eState));
        f_MessageSet(_stMsg);
      END_IF
    END_IF
END_CASE
CASE _eState
OF
  E_PROGRESS.PROGRESS_WORKING:
    _eState                         := E_PROGRESS.PROGRESS_STILL_WORKING;
    _nNumPointsRead                 := TO_UINT(_fbReadMotionFunction.NumPointsRead);
    _nMotionFunctionSize            := SEL((TO_UINT(_mcCamRef.ArraySize) > MAX_MOTION_FUNCTION_POINTS),
                                            TO_UINT(_mcCamRef.ArraySize),
                                            MAX_MOTION_FUNCTION_POINTS);

    memcpy(ADR(_mcMotionFunction), _mcCamRef.pArray, _nMotionFunctionSize); 

    _stMsg.eType                    := SEL((TO_UINT(_mcCamRef.ArraySize) > MAX_MOTION_FUNCTION_POINTS),
                                            E_MessageType.eMessageInfo,
                                            E_MessageType.eMessageWarning);

    _stMsg.eDevice                  := E_Device.Camming + (_AxisSlave.NcToPlc.AxisId);
    _stMsg.eSubdevice               := e_Subdevice.fbReadMotionFunction;
    _stMsg.iErrorNumber             := _nMotionFunctionSize;

    _stMsg.sText                    := concat(' : ', TO_STRING(_eState));

    IF (_MessageLevel > E_MessageType.eMessageError)
    THEN
      f_MessageSet(_stMsg);
    END_IF

END_CASE
CASE _eState
OF
  E_PROGRESS.PROGRESS_STILL_WORKING:
    _eState                         := E_PROGRESS.PROGRESS_DONE;

(*
    _stMotionFunction.stMotionFunction    := _mcMotionFunction;
    _stMotionFunction.nMotionFunctionSize := _nMotionFunctionSize;
    _stMotionFunction.nPoints             := TO_UINT(_fbReadMotionFunction.NumPointsRead);
*)

    IF (_MessageLevel > E_MessageType.eMessageError)
    THEN
      _stMsg.eType                  := E_MessageType.eMessageInfo;
      _stMsg.eDevice                := E_Device.Camming + (_AxisSlave.NcToPlc.AxisId);
      _stMsg.eSubdevice             := e_Subdevice.fbReadMotionFunction;
      _stMsg.iErrorNumber           := 0;
  
      _stMsg.sText                  := concat(' : ', TO_STRING(_eState));
      f_MessageSet(_stMsg);
    END_IF

    _fbReadMotionFunction(
              Execute               := FALSE, 
              CamTableID            := _stCamData.nCamTableId, 
              PointID               := _stCamData.nPointId, 
              NumPoints             := _stCamData.nNumPoints, 
              CamTable              := _mcCamRef);
END_CASE

ReadMotionFunction                  := _eState;
END_METHOD

PROPERTY ReadMotionFunctionData : ST_MOTION_FUNCTION
GET
VAR
  _idx        : UINT;
  _stMf       : ST_MOTION_FUNCTION;
END_VAR

_stMf.nMotionFunctionSize   := TO_UINT(_mcCamRef.ArraySize);
_stMf.nPoints               := TO_UINT(_mcCamRef.NoOfRows);

FOR _idx := 1 TO MAX_MOTION_FUNCTION_POINTS
DO
  IF NOT (_idx > _stMf.nPoints)
  THEN
    _stMf.stMotionFunction[_idx].nFunctionType      := TO_UINT(_mcMotionFunction[_idx].FunctionType);
    _stMf.stMotionFunction[_idx].nPointIndex        := TO_UINT(_mcMotionFunction[_idx].PointIndex);
    _stMf.stMotionFunction[_idx].nRelIndexNextPoint := TO_UINT(_mcMotionFunction[_idx].RelIndexNextPoint);

    _stMf.stMotionFunction[_idx].wPointType         := TO_WORD(_mcMotionFunction[_idx].PointType);

    _stMf.stMotionFunction[_idx].rMasterPos         := _mcMotionFunction[_idx].MasterPos;
    _stMf.stMotionFunction[_idx].rSlavePos          := _mcMotionFunction[_idx].SlavePos;

    _stMf.stMotionFunction[_idx].rSlaveVelo         := _mcMotionFunction[_idx].SlaveVelo;
    _stMf.stMotionFunction[_idx].rSlaveAcc          := _mcMotionFunction[_idx].SlaveAcc;
    _stMf.stMotionFunction[_idx].rSlaveJerk         := _mcMotionFunction[_idx].SlaveJerk;
  END_IF
END_FOR

ReadMotionFunctionData := _stMf;
END_GET
END_PROPERTY

METHOD ReadMotionFunctionPoint : E_PROGRESS
VAR_INPUT
  Execute           : BOOL;
END_VAR
VAR_INST
  _eState           : E_PROGRESS;
  _rValue           : LREAL;
  _udiErr           : UDINT;
  _stMsg            : ST_Message;
END_VAR

IF NOT Execute THEN _eState   := E_PROGRESS.PROGRESS_INIT; END_IF


CASE _eState
OF
  E_PROGRESS.PROGRESS_INIT:
    IF Execute 
    THEN
      memset(ADR(_mcMotionFunctionPoint),0,SIZEOF(_mcMotionFunctionPoint));
      memset(ADR(_stMsg),0,SIZEOF(_stMsg));
      _udiErr                       := 0;
      _rValue                       := 0;
      _eState                       := E_PROGRESS.PROGRESS_BUSY;

      _fbReadMotionFunctionPoint(
              Execute               := FALSE, 
              CamTableID            := _stCamData.nCamTableId, 
              PointID               := _stCamData.nPointId,
              Point                 := _mcMotionFunctionPoint);
    END_IF
END_CASE
CASE _eState
OF
  E_PROGRESS.PROGRESS_BUSY:
    _fbReadMotionFunctionPoint(
              Execute               := TRUE, 
              CamTableID            := _stCamData.nCamTableId, 
              PointID               := _stCamData.nPointId,
              Point                 := _mcMotionFunctionPoint);

    IF (_fbReadMotionFunctionPoint.Error)
    THEN
      _eState                       := E_PROGRESS.PROGRESS_ERROR;
      _udiErr                       := _fbReadMotionFunctionPoint.ErrorID;

      _stMsg.eType                  := E_MessageType.eMessageError;
      _stMsg.eDevice                := E_Device.Camming + (_AxisSlave.NcToPlc.AxisId);
      _stMsg.eSubdevice             := e_Subdevice.fbReadMotionFunctionPoint;
      _stMsg.iErrorNumber           := _udiErr;

      _stMsg.sText                  := concat(' : ', TO_STRING(_eState));
      f_MessageSet(_stMsg);

      _fbReadMotionFunctionPoint(
              Execute               := FALSE, 
              CamTableID            := _stCamData.nCamTableId, 
              PointID               := _stCamData.nPointId,
              Point                 := _mcMotionFunctionPoint);
    ELSE
      IF (_fbReadMotionFunctionPoint.Done)
      THEN
        _eState                     := E_PROGRESS.PROGRESS_DONE;
  
        _stMsg.eType                := E_MessageType.eMessageInfo;
        _stMsg.eDevice              := E_Device.Camming + (_AxisSlave.NcToPlc.AxisId);
        _stMsg.eSubdevice           := e_Subdevice.fbReadMotionFunctionPoint;
        _stMsg.iErrorNumber         := 0;
  
        _stMsg.sText                := concat(' : ', TO_STRING(_eState));

        IF (_MessageLevel > E_MessageType.eMessageError)
        THEN
          f_MessageSet(_stMsg);
        END_IF

        _fbReadMotionFunctionPoint(
              Execute               := FALSE, 
              CamTableID            := _stCamData.nCamTableId, 
              PointID               := _stCamData.nPointId,
              Point                 := _mcMotionFunctionPoint);
      END_IF
    END_IF
END_CASE

ReadMotionFunctionPoint             := _eState;
END_METHOD

PROPERTY ReadMotionFunctionPointData : ST_MOTION_FUNCTION_POINT
GET
VAR
  _stTmp    : ST_MOTION_FUNCTION_POINT;
END_VAR

_stTmp.nFunctionType        := TO_UINT(_mcMotionFunctionPoint.FunctionType);
_stTmp.nPointIndex          := TO_UINT(_mcMotionFunctionPoint.PointIndex);
_stTmp.nRelIndexNextPoint   := TO_UINT(_mcMotionFunctionPoint.RelIndexNextPoint);
_stTmp.wPointType           := TO_WORD(_mcMotionFunctionPoint.PointType);

_stTmp.rMasterPos           := _mcMotionFunctionPoint.MasterPos;
_stTmp.rSlavePos            := _mcMotionFunctionPoint.SlavePos;
_stTmp.rSlaveAcc            := _mcMotionFunctionPoint.SlaveAcc;
_stTmp.rSlaveJerk           := _mcMotionFunctionPoint.SlaveJerk;
_stTmp.rSlaveVelo           := _mcMotionFunctionPoint.SlaveVelo;

ReadMotionFunctionPointData := _stTmp;
END_GET
END_PROPERTY

METHOD ReadMotionFunctionValues : E_PROGRESS
VAR_INPUT
  Execute           : BOOL;
END_VAR
VAR_INST
  _eState           : E_PROGRESS;
  _rValue           : LREAL;
  _udiErr           : UDINT;
  _stMsg            : ST_Message;
END_VAR

IF NOT Execute THEN _eState   := E_PROGRESS.PROGRESS_INIT; END_IF


CASE _eState
OF
  E_PROGRESS.PROGRESS_INIT:
    IF Execute 
    THEN
      memset(ADR(_mcMotionFunction),0,SIZEOF(_mcMotionFunction));
      memset(ADR(_stMsg),0,SIZEOF(_stMsg));
      _udiErr                       := 0;
      _rValue                       := 0;
      _eState                       := E_PROGRESS.PROGRESS_BUSY;

      _mcCamRef.pArray              := ADR(_mcMotionFunction);
      _mcCamRef.ArraySize           := SIZEOF(_mcMotionFunction);

      _mcCamRef.TableType           := Tc2_MC2_Camming.MC_TABLETYPE_MOTIONFUNCTION;
      _mcCamRef.NoOfColumns         := 1;

      _fbReadMotionFunctionValues(
              Execute               := FALSE, 
              CamTableID            := _stCamData.nCamTableId, 
              ValueSelectMask       := _stCamData.stReadValuesParameter.nValueSelectMask, 
              StartPosMaster        := _stCamData.stReadValuesParameter.rValueMasterStart, 
              EndPosMaster          := _stCamData.stReadValuesParameter.rValueMasterEnd, 
              Increment             := _stCamData.stReadValuesParameter.rIncrement, 
              CamTable              := _mcCamRef);
    END_IF
END_CASE
CASE _eState
OF
  E_PROGRESS.PROGRESS_BUSY:
    _fbReadMotionFunctionValues(
              Execute               := TRUE, 
              CamTableID            := _stCamData.nCamTableId, 
              ValueSelectMask       := _stCamData.stReadValuesParameter.nValueSelectMask, 
              StartPosMaster        := _stCamData.stReadValuesParameter.rValueMasterStart, 
              EndPosMaster          := _stCamData.stReadValuesParameter.rValueMasterEnd, 
              Increment             := _stCamData.stReadValuesParameter.rIncrement, 
              CamTable              := _mcCamRef);

    IF (_fbReadMotionFunctionValues.Error)
    THEN
      _eState                       := E_PROGRESS.PROGRESS_ERROR;
      _udiErr                       := _fbReadMotionFunctionValues.ErrorID;

      _stMsg.eType                  := E_MessageType.eMessageError;
      _stMsg.eDevice                := E_Device.Camming + (_AxisSlave.NcToPlc.AxisId);
      _stMsg.eSubdevice             := e_Subdevice.fbReadMotionFunctionValues;
      _stMsg.iErrorNumber           := _udiErr;

      _stMsg.sText                  := concat(' : ', TO_STRING(_eState));
      f_MessageSet(_stMsg);

      _fbReadMotionFunctionValues(
              Execute               := FALSE, 
              CamTableID            := _stCamData.nCamTableId, 
              ValueSelectMask       := _stCamData.stReadValuesParameter.nValueSelectMask, 
              StartPosMaster        := _stCamData.stReadValuesParameter.rValueMasterStart, 
              EndPosMaster          := _stCamData.stReadValuesParameter.rValueMasterEnd, 
              Increment             := _stCamData.stReadValuesParameter.rIncrement, 
              CamTable              := _mcCamRef);
    ELSE
      IF (_fbReadMotionFunctionValues.Done)
      THEN
        _eState                     := E_PROGRESS.PROGRESS_DONE;
  
        _stMsg.eType                := E_MessageType.eMessageInfo;
        _stMsg.eDevice              := E_Device.Camming + (_AxisSlave.NcToPlc.AxisId);
        _stMsg.eSubdevice           := e_Subdevice.fbReadMotionFunctionValues;
        _stMsg.iErrorNumber         := 0;
  
        _stMsg.sText                := concat(' : ', TO_STRING(_eState));

        IF (_MessageLevel > E_MessageType.eMessageError)
        THEN
          f_MessageSet(_stMsg);
        END_IF
        _fbReadMotionFunctionValues(
              Execute               := FALSE, 
              CamTableID            := _stCamData.nCamTableId, 
              ValueSelectMask       := _stCamData.stReadValuesParameter.nValueSelectMask, 
              StartPosMaster        := _stCamData.stReadValuesParameter.rValueMasterStart, 
              EndPosMaster          := _stCamData.stReadValuesParameter.rValueMasterEnd, 
              Increment             := _stCamData.stReadValuesParameter.rIncrement, 
              CamTable              := _mcCamRef);
      END_IF
    END_IF
END_CASE

ReadMotionFunctionValues            := _eState;
END_METHOD

METHOD SetOnLineChangeMode : E_PROGRESS
VAR_INPUT
  Execute           : BOOL;
END_VAR
VAR_INST
  _eState           : E_PROGRESS;
  _rValue           : LREAL;
  _udiErr           : UDINT;
  _stMsg            : ST_Message;

  _nCopySize        : UINT;

END_VAR

IF NOT Execute THEN _eState   := E_PROGRESS.PROGRESS_INIT; END_IF


CASE _eState
OF
  E_PROGRESS.PROGRESS_INIT:
    IF Execute 
    THEN
      memset(ADR(_stMsg),0,SIZEOF(_stMsg));
      _udiErr                       := 0;
      _rValue                       := 0;
      _eState                       := E_PROGRESS.PROGRESS_BUSY;

      _fbSetCamOnlineChangeMode(
              Execute               := FALSE, 
              ActivationMode        := _stCamData.nActivationMode, 
              ActivationPosition    := _stCamData.rActivationPosition, 
              MasterScalingMode     := _stCamData.stCamScalingData.nMasterScalingMode, 
              SlaveScalingMode      := _stCamData.stCamScalingData.nSlaveScalingMode, 
              CamTableID            := _stCamData.nCamTableId);
    END_IF
END_CASE
CASE _eState
OF
  E_PROGRESS.PROGRESS_BUSY:
    _fbSetCamOnlineChangeMode(
              Execute               := TRUE, 
              ActivationMode        := _stCamData.nActivationMode, 
              ActivationPosition    := _stCamData.rActivationPosition, 
              MasterScalingMode     := _stCamData.stCamScalingData.nMasterScalingMode, 
              SlaveScalingMode      := _stCamData.stCamScalingData.nSlaveScalingMode, 
              CamTableID            := _stCamData.nCamTableId);

    IF (_fbSetCamOnlineChangeMode.Error)
    THEN
      _eState                       := E_PROGRESS.PROGRESS_ERROR;
      _udiErr                       := _fbSetCamOnlineChangeMode.ErrorID;

      _stMsg.eType                  := E_MessageType.eMessageError;
      _stMsg.eDevice                := E_Device.Camming + (_AxisSlave.NcToPlc.AxisId);
      _stMsg.eSubdevice             := e_Subdevice.fbSetOnlineChangeMode;
      _stMsg.iErrorNumber           := _udiErr;

      _stMsg.sText                  := concat(' : ', TO_STRING(_eState));
      f_MessageSet(_stMsg);

      _fbSetCamOnlineChangeMode(
              Execute               := FALSE); 

    ELSIF (_fbSetCamOnlineChangeMode.Done)
    THEN
      _eState                       := E_PROGRESS.PROGRESS_DONE;

      _stMsg.eType                  := E_MessageType.eMessageInfo;
      _stMsg.eDevice                := E_Device.Camming + (_AxisSlave.NcToPlc.AxisId);
      _stMsg.eSubdevice             := e_Subdevice.fbSetOnlineChangeMode;
      _stMsg.iErrorNumber           := 0;

      _stMsg.sText                  := concat(' : ', TO_STRING(_eState));

      IF (_MessageLevel > E_MessageType.eMessageError)
      THEN
        f_MessageSet(_stMsg);
      END_IF

      _fbSetCamOnlineChangeMode(
              Execute               := FALSE); 
    END_IF
END_CASE

SetOnLineChangeMode                 := _eState;
END_METHOD

METHOD WriteMotionFunction : E_PROGRESS
VAR_INPUT
  Execute           : BOOL;
END_VAR
VAR_INST
  _eResult,
  _eState           : E_PROGRESS;
  _rValue           : LREAL;
  _udiErr           : UDINT;
  _stMsg            : ST_Message;


END_VAR
IF NOT __ISVALIDREF(_AxisSlave)
THEN
  _eCheck                     := E_CHECK_STATE.CAM_SLAVE_AXIS_REF_INVALID;
  WriteMotionFunction         := E_PROGRESS.PROGRESS_ERROR;
  RETURN;
END_IF

IF NOT Execute THEN _eState := E_PROGRESS.PROGRESS_INIT; END_IF

CASE _eState
OF
  E_PROGRESS.PROGRESS_INIT:
    IF Execute 
    THEN
      memset(ADR(_stMsg),0,SIZEOF(_stMsg));
      _udiErr                       := 0;
      _rValue                       := 0;
      _eState                       := E_PROGRESS.PROGRESS_BUSY;
      _eResult                      := SetOnLineChangeMode(FALSE);
    END_IF
END_CASE
CASE _eState
OF
  E_PROGRESS.PROGRESS_BUSY:
    _eResult                        := SetOnLineChangeMode(TRUE);
    IF (_eResult = E_PROGRESS.PROGRESS_ERROR)
    THEN
      SetOnLineChangeMode(FALSE);
      _eState                       := E_PROGRESS.PROGRESS_ERROR;
    ELSE
      IF (_eResult = E_PROGRESS.PROGRESS_DONE)
      THEN
        SetOnLineChangeMode(FALSE);
        _eState                     := E_PROGRESS.PROGRESS_STARTUP;
(*
        _mcMotionFunction           := _stMotionFunction.stMotionFunction;
*)
      END_IF
    END_IF
END_CASE
CASE _eState
OF
  E_PROGRESS.PROGRESS_STARTUP:
    _eState                         := E_PROGRESS.PROGRESS_WORKING;

    _mcCamRef.pArray                := ADR(_mcMotionFunction);
    _mcCamRef.ArraySize             := SIZEOF(_mcMotionFunction);

    _mcCamRef.TableType             := Tc2_MC2_Camming.MC_TABLETYPE_MOTIONFUNCTION;
    _mcCamRef.NoOfColumns           := 1;

    _fbWriteMotionFunction(
                    Execute         := FALSE, 
                    CamTableID      := _stCamData.nCamTableId, 
                    PointID         := _stCamData.nPointId, 
                    NumPoints       := _stCamData.nNumPoints, 
                    CamTable        := _mcCamRef);

END_CASE
CASE _eState
OF
  E_PROGRESS.PROGRESS_WORKING:
    _fbWriteMotionFunction(
                    Execute         := TRUE, 
                    CamTableID      := _stCamData.nCamTableId, 
                    PointID         := _stCamData.nPointId, 
                    NumPoints       := _stCamData.nNumPoints, 
                    CamTable        := _mcCamRef);

    IF (_fbWriteMotionFunction.Error)
    THEN
      _eState                       := E_PROGRESS.PROGRESS_ERROR;
      _udiErr                       := _fbWriteMotionFunction.ErrorID;

      _stMsg.eType                  := E_MessageType.eMessageError;
      _stMsg.eDevice                := E_Device.Camming + (_AxisSlave.NcToPlc.AxisId);
      _stMsg.eSubdevice             := e_Subdevice.fbWriteMotionFunction;
      _stMsg.iErrorNumber           := _udiErr;

      _stMsg.sText                  := concat(' : ', TO_STRING(_eState));
      f_MessageSet(_stMsg);

      _fbWriteMotionFunction(
                    Execute         := FALSE, 
                    CamTableID      := _stCamData.nCamTableId, 
                    PointID         := _stCamData.nPointId, 
                    NumPoints       := _stCamData.nNumPoints, 
                    CamTable        := _mcCamRef);
    ELSE
      IF (_fbWriteMotionFunction.Done)
      THEN
        _eState                     := E_PROGRESS.PROGRESS_STILL_WORKING;
        _fbWriteMotionFunction(
                    Execute         := FALSE, 
                    CamTableID      := _stCamData.nCamTableId, 
                    PointID         := _stCamData.nPointId, 
                    NumPoints       := _stCamData.nNumPoints, 
                    CamTable        := _mcCamRef);
      END_IF
    END_IF
END_CASE
CASE _eState
OF
  E_PROGRESS.PROGRESS_STILL_WORKING:
    _eState                         := E_PROGRESS.PROGRESS_DONE;

    _stMsg.eType                    := E_MessageType.eMessageInfo;
    _stMsg.eDevice                  := E_Device.Camming + (_AxisSlave.NcToPlc.AxisId);
    _stMsg.eSubdevice               := e_Subdevice.fbWriteMotionFunction;
    _stMsg.iErrorNumber             := 0;

    _stMsg.sText                    := concat(' : ', TO_STRING(_eState));

    IF (_MessageLevel > E_MessageType.eMessageError)
    THEN
      f_MessageSet(_stMsg);
    END_IF
END_CASE

WriteMotionFunction                 := _eState;
END_METHOD

PROPERTY WriteMotionFunctionData : ST_MOTION_FUNCTION
SET
VAR
  _idx        : UINT;
  _stMf       : ST_MOTION_FUNCTION;
END_VAR

_stMf                                           := WriteMotionFunctionData;
memset(ADR(_mcMotionFunction), 0, SIZEOF(_mcMotionFunction));

FOR _idx := 1 TO MAX_MOTION_FUNCTION_POINTS
DO
  IF NOT (_idx > _stMf.nPoints)
  THEN
    _mcMotionFunction[_idx].FunctionType        := TO_INT(_stMf.stMotionFunction[_idx].nFunctionType);
    _mcMotionFunction[_idx].PointIndex          := _stMf.stMotionFunction[_idx].nPointIndex;
    _mcMotionFunction[_idx].RelIndexNextPoint   := _stMf.stMotionFunction[_idx].nRelIndexNextPoint;

    _mcMotionFunction[_idx].PointType           := to_int(_stMf.stMotionFunction[_idx].wPointType);

    _mcMotionFunction[_idx].MasterPos           := _stMf.stMotionFunction[_idx].rMasterPos;
    _mcMotionFunction[_idx].SlavePos            := _stMf.stMotionFunction[_idx].rSlavePos;

    _mcMotionFunction[_idx].SlaveVelo           := _stMf.stMotionFunction[_idx].rSlaveVelo;
    _mcMotionFunction[_idx].SlaveAcc            := _stMf.stMotionFunction[_idx].rSlaveAcc;
    _mcMotionFunction[_idx].SlaveJerk           := _stMf.stMotionFunction[_idx].rSlaveJerk;
  END_IF
END_FOR
END_SET
END_PROPERTY

METHOD WriteMotionFunctionPoint : E_PROGRESS
VAR_INPUT
  Execute           : BOOL;
END_VAR
VAR_INST
  _eResult,
  _eState           : E_PROGRESS;
  _rValue           : LREAL;
  _udiErr           : UDINT;
  _stMsg            : ST_Message;


END_VAR
IF NOT __ISVALIDREF(_AxisSlave)
THEN
  _eCheck                     := E_CHECK_STATE.CAM_SLAVE_AXIS_REF_INVALID;
  WriteMotionFunctionPoint    := E_PROGRESS.PROGRESS_ERROR;
  RETURN;
END_IF

IF NOT Execute THEN _eState := E_PROGRESS.PROGRESS_INIT; END_IF

CASE _eState
OF
  E_PROGRESS.PROGRESS_INIT:
    IF Execute 
    THEN
      memset(ADR(_stMsg),0,SIZEOF(_stMsg));
      _udiErr                       := 0;
      _rValue                       := 0;
      _eState                       := E_PROGRESS.PROGRESS_BUSY;
      _eResult                      := SetOnLineChangeMode(FALSE);

      IF (_stCamData.nPointIndex < 1) OR
         (_stCamData.nPointIndex > MAX_MOTION_FUNCTION_POINTS)
      THEN
        _eState                     := E_PROGRESS.PROGRESS_ERROR;
        _udiErr                     := _stCamData.nPointIndex;
  
        _stMsg.eType                := E_MessageType.eMessageError;
        _stMsg.eDevice              := E_Device.Camming + (_AxisSlave.NcToPlc.AxisId);
        _stMsg.eSubdevice           := e_Subdevice.fbWriteMotionFunctionPoint;
        _stMsg.iErrorNumber         := _udiErr;
  
        _stMsg.sText                  := concat('POINT INDEX NOT IN RANGE: ', TO_STRING(_eState));
        f_MessageSet(_stMsg);

      END_IF
    END_IF
END_CASE
CASE _eState
OF
  E_PROGRESS.PROGRESS_BUSY:
    _eResult                        := SetOnLineChangeMode(TRUE);
    IF (_eResult = E_PROGRESS.PROGRESS_ERROR)
    THEN
      SetOnLineChangeMode(FALSE);
      _eState                       := E_PROGRESS.PROGRESS_ERROR;
    ELSE
      IF (_eResult = E_PROGRESS.PROGRESS_DONE)
      THEN
        SetOnLineChangeMode(FALSE);
        _eState                     := E_PROGRESS.PROGRESS_STARTUP;
(*
        _mcMotionFunction           := _stMotionFunction.stMotionFunction;
*)
        _mcMotionFunctionPoint      := _mcMotionFunction[_stCamData.nPointIndex];
      END_IF
    END_IF
END_CASE
CASE _eState
OF
  E_PROGRESS.PROGRESS_STARTUP:
    _eState                         := E_PROGRESS.PROGRESS_WORKING;
    _fbWriteMotionFunctionPoint(
                      Execute       := FALSE, 
                      CamTableID    := _stCamData.nCamTableId, 
                      PointID       := _stCamData.nPointId,
                      Point         := _mcMotionFunctionPoint);
END_CASE
CASE _eState
OF
  E_PROGRESS.PROGRESS_WORKING:
    _fbWriteMotionFunctionPoint(
                      Execute       := TRUE, 
                      CamTableID    := _stCamData.nCamTableId, 
                      PointID       := _stCamData.nPointId,
                      Point         := _mcMotionFunctionPoint);

    IF (_fbWriteMotionFunctionPoint.Error)
    THEN
      _eState                       := E_PROGRESS.PROGRESS_ERROR;
      _udiErr                       := _fbWriteMotionFunctionPoint.ErrorID;

      _stMsg.eType                  := E_MessageType.eMessageError;
      _stMsg.eDevice                := E_Device.Camming + (_AxisSlave.NcToPlc.AxisId);
      _stMsg.eSubdevice             := e_Subdevice.fbWriteMotionFunctionPoint;
      _stMsg.iErrorNumber           := _udiErr;

      _stMsg.sText                  := concat(' : ', TO_STRING(_eState));
      f_MessageSet(_stMsg);

      _fbWriteMotionFunctionPoint(
                      Execute       := FALSE, 
                      CamTableID    := _stCamData.nCamTableId, 
                      PointID       := _stCamData.nPointId,
                      Point         := _mcMotionFunctionPoint);

    ELSE
      IF (_fbWriteMotionFunctionPoint.Done)
      THEN
        _eState                     := E_PROGRESS.PROGRESS_STILL_WORKING;
        _fbWriteMotionFunctionPoint(
                      Execute       := FALSE, 
                      CamTableID    := _stCamData.nCamTableId, 
                      PointID       := _stCamData.nPointId,
                      Point         := _mcMotionFunctionPoint);
      END_IF
    END_IF
END_CASE
CASE _eState
OF
  E_PROGRESS.PROGRESS_STILL_WORKING:
    _eState                         := E_PROGRESS.PROGRESS_DONE;

    _stMsg.eType                    := E_MessageType.eMessageInfo;
    _stMsg.eDevice                  := E_Device.Camming + (_AxisSlave.NcToPlc.AxisId);
    _stMsg.eSubdevice               := e_Subdevice.fbWriteMotionFunctionPoint;
    _stMsg.iErrorNumber             := 0;

    _stMsg.sText                    := concat(' : ', TO_STRING(_eState));

    IF (_MessageLevel > E_MessageType.eMessageError)
    THEN
      f_MessageSet(_stMsg);
    END_IF
END_CASE

WriteMotionFunctionPoint            := _eState;
END_METHOD

PROPERTY WriteMotionFunctionPointData : ST_MOTION_FUNCTION_POINT
SET
VAR
  _idx        : UINT;
  _stMf       : ST_MOTION_FUNCTION_POINT;
END_VAR

_stMf                                       := WriteMotionFunctionPointData;
memset(ADR(_mcMotionFunctionPoint), 0, SIZEOF(_mcMotionFunctionPoint));

_mcMotionFunctionPoint.FunctionType         := TO_INT(_stMf.nFunctionType);
_mcMotionFunctionPoint.PointIndex           := _stMf.nPointIndex;
_mcMotionFunctionPoint.RelIndexNextPoint    := _stMf.nRelIndexNextPoint;

_mcMotionFunctionPoint.PointType            := TO_INT(_stMf.wPointType);

_mcMotionFunctionPoint.MasterPos            := _stMf.rMasterPos;
_mcMotionFunctionPoint.SlavePos             := _stMf.rSlavePos;

_mcMotionFunctionPoint.SlaveVelo            := _stMf.rSlaveVelo;
_mcMotionFunctionPoint.SlaveAcc             := _stMf.rSlaveAcc;
_mcMotionFunctionPoint.SlaveJerk            := _stMf.rSlaveJerk;
END_SET
END_PROPERTY

END_FUNCTION_BLOCK

